LIN {X 0,Y 198.833,Z 382.031,A -85,B 0,C 180,E1 -24400.179,E2 -24400.179} C_VEL
LIN {X 0,Y 188.917,Z 377.763,A -85,B 0,C 180,E1 -24404.769,E2 -24404.769} C_VEL
LIN {X 0,Y 183.38,Z 374.333,A -85,B 0,C 180,E1 -24407.854,E2 -24407.854} C_VEL
LIN {X 0,Y 177.292,Z 368.639,A -85,B 0,C 180,E1 -24412.116,E2 -24412.116} C_VEL
LIN {X 0,Y 173.181,Z 362.778,A -85,B 0,C 180,E1 -24415.87,E2 -24415.87} C_VEL
LIN {X 0,Y 170.579,Z 356.861,A -85,B 0,C 180,E1 -24419.135,E2 -24419.135} C_VEL
LIN {X 0,Y 168.518,Z 348.975,A -85,B 0,C 180,E1 -24422.83,E2 -24422.83} C_VEL
LIN {X 0,Y 167.275,Z 340.992,A -85,B 0,C 180,E1 -24426.029,E2 -24426.029} C_VEL
LIN {X 0,Y 165.67,Z 333.745,A -85,B 0,C 180,E1 -24428.814,E2 -24428.814} C_VEL
LIN {X 0,Y 163.533,Z 326.252,A -85,B 0,C 180,E1 -24431.653,E2 -24431.653} C_VEL
LIN {X 0,Y 160.686,Z 318.576,A -85,B 0,C 180,E1 -24434.641,E2 -24434.641} C_VEL
LIN {X 0,Y 156.368,Z 309.383,A -85,B 0,C 180,E1 -24438.458,E2 -24438.458} C_VEL
LIN {X 0,Y 152.513,Z 302.543,A -85,B 0,C 180,E1 -24441.569,E2 -24441.569} C_VEL
LIN {X 0,Y 150.34,Z 299.173,A -85,B 0,C 180,E1 -24443.332,E2 -24443.332} C_VEL
LIN {X 0,Y 149.453,Z 297.828,A -85,B 0,C 180,E1 -24444.02,E2 -24444.02} C_VEL
LIN {X 0,Y 147.324,Z 294.974,A -85,B 0,C 180,E1 -24445.691,E2 -24445.691} C_VEL
LIN {X 0,Y 146.51,Z 293.362,A -85,B 0,C 180,E1 -24446.457,E2 -24446.457} C_VEL
LIN {X 0,Y 144.109,Z 290.974,A -85,B 0,C 180,E1 -24448.403,E2 -24448.403} C_VEL
LIN {X 0,Y 143.178,Z 288.494,A -85,B 0,C 180,E1 -24449.406,E2 -24449.406} C_VEL
LIN {X 0,Y 143.104,Z 288.159,A -85,B 0,C 180,E1 -24449.593,E2 -24449.593} C_VEL
LIN {X 0,Y 143.128,Z 288.151,A -85,B 0,C 180,E1 -24453.793,E2 -24453.793} C_VEL
LIN {X 0,Y 143.229,Z 288.133,A -85,B 0,C 180,E1 -24459.93,E2 -24459.93} C_VEL
LIN {X 0,Y 143.298,Z 288.126,A -85,B 0,C 180,E1 -24465.823,E2 -24465.823} C_VEL
LIN {X 0,Y 143.521,Z 288.105,A -85,B 0,C 180,E1 -24468.722,E2 -24468.722} C_VEL
LIN {X 0,Y 143.611,Z 288.09,A -85,B 0,C 180,E1 -24471.575,E2 -24471.575} C_VEL
LIN {X 0,Y 144.158,Z 287.993,A -85,B 0,C 180,E1 -24480.016,E2 -24480.016} C_VEL
LIN {X 0,Y 143.622,Z 288.096,A -85,B 0,C 180,E1 -24488.458,E2 -24488.458} C_VEL
LIN {X 0,Y 143.504,Z 288.112,A -85,B 0,C 180,E1 -24491.633,E2 -24491.633} C_VEL
LIN {X 0,Y 143.247,Z 288.145,A -85,B 0,C 180,E1 -24497.136,E2 -24497.136} C_VEL
LIN {X 0,Y 143.35,Z 288.954,A -85,B 0,C 180,E1 -24501.332,E2 -24501.332} C_VEL
LIN {X 0,Y 143.471,Z 290.546,A -85,B 0,C 180,E1 -24508.15,E2 -24508.15} C_VEL
LIN {X 0,Y 143.582,Z 291.452,A -85,B 0,C 180,E1 -24510.74,E2 -24510.74} C_VEL
LIN {X 0,Y 144.635,Z 294.391,A -85,B 0,C 180,E1 -24511.814,E2 -24511.814} C_VEL
LIN {X 0,Y 147.362,Z 297.867,A -85,B 0,C 180,E1 -24514.044,E2 -24514.044} C_VEL
LIN {X 0,Y 148.991,Z 301.335,A -85,B 0,C 180,E1 -24515.523,E2 -24515.523} C_VEL
LIN {X 0,Y 150.405,Z 303.365,A -85,B 0,C 180,E1 -24516.585,E2 -24516.585} C_VEL
LIN {X 0,Y 152.587,Z 307.744,A -85,B 0,C 180,E1 -24518.465,E2 -24518.465} C_VEL
LIN {X 0,Y 155.821,Z 315.822,A -85,B 0,C 180,E1 -24521.485,E2 -24521.485} C_VEL
LIN {X 0,Y 158.01,Z 323.997,A -85,B 0,C 180,E1 -24524.218,E2 -24524.218} C_VEL
LIN {X 0,Y 159.377,Z 333.893,A -85,B 0,C 180,E1 -24527.295,E2 -24527.295} C_VEL
LIN {X 0,Y 159.634,Z 344.227,A -85,B 0,C 180,E1 -24530.573,E2 -24530.573} C_VEL
LIN {X 0,Y 159.227,Z 352.071,A -85,B 0,C 180,E1 -24533.24,E2 -24533.24} C_VEL
LIN {X 0,Y 158.008,Z 360.113,A -85,B 0,C 180,E1 -24536.222,E2 -24536.222} C_VEL
LIN {X 0,Y 154.348,Z 367.945,A -85,B 0,C 180,E1 -24539.187,E2 -24539.187} C_VEL
LIN {X 0,Y 151.04,Z 374.482,A -85,B 0,C 180,E1 -24542.271,E2 -24542.271} C_VEL
LIN {X 0,Y 148.752,Z 378.986,A -85,B 0,C 180,E1 -24544.836,E2 -24544.836} C_VEL
LIN {X 0,Y 145.708,Z 384.478,A -85,B 0,C 180,E1 -24548.793,E2 -24548.793} C_VEL
LIN {X 0,Y 143.303,Z 388.804,A -85,B 0,C 180,E1 -24552.887,E2 -24552.887} C_VEL
LIN {X 0,Y 142.229,Z 391.177,A -85,B 0,C 180,E1 -24555.696,E2 -24555.696} C_VEL
LIN {X 0,Y 141.418,Z 392.982,A -85,B 0,C 180,E1 -24558.534,E2 -24558.534} C_VEL
LIN {X 0,Y 140.571,Z 395.441,A -85,B 0,C 180,E1 -24564.261,E2 -24564.261} C_VEL
LIN {X 0,Y 140.517,Z 396.037,A -85,B 0,C 180,E1 -24567.133,E2 -24567.133} C_VEL
LIN {X 0,Y 140.592,Z 396.196,A -85,B 0,C 180,E1 -24570,E2 -24570} C_VEL
LIN {X 0,Y 140.517,Z 396.037,A -85,B 0,C 180,E1 -24572.867,E2 -24572.867} C_VEL
LIN {X 0,Y 140.57,Z 395.441,A -85,B 0,C 180,E1 -24575.739,E2 -24575.739} C_VEL
LIN {X 0,Y 141.391,Z 392.981,A -85,B 0,C 180,E1 -24581.468,E2 -24581.468} C_VEL
LIN {X 0,Y 142.734,Z 390.024,A -85,B 0,C 180,E1 -24585.712,E2 -24585.712} C_VEL
LIN {X 0,Y 144.826,Z 386.032,A -85,B 0,C 180,E1 -24589.857,E2 -24589.857} C_VEL
LIN {X 0,Y 147.624,Z 380.901,A -85,B 0,C 180,E1 -24593.869,E2 -24593.869} C_VEL
LIN {X 0,Y 150.517,Z 375.641,A -85,B 0,C 180,E1 -24597.08,E2 -24597.08} C_VEL
LIN {X 0,Y 153.589,Z 369.319,A -85,B 0,C 180,E1 -24600.221,E2 -24600.221} C_VEL
LIN {X 0,Y 156.521,Z 363.369,A -85,B 0,C 180,E1 -24602.602,E2 -24602.602} C_VEL
LIN {X 0,Y 157.965,Z 360.112,A -85,B 0,C 180,E1 -24603.788,E2 -24603.788} C_VEL
LIN {X 0,Y 159.233,Z 352.131,A -85,B 0,C 180,E1 -24606.735,E2 -24606.735} C_VEL
LIN {X 0,Y 159.664,Z 342.122,A -85,B 0,C 180,E1 -24610.113,E2 -24610.113} C_VEL
LIN {X 0,Y 159.16,Z 332.099,A -85,B 0,C 180,E1 -24613.25,E2 -24613.25} C_VEL
LIN {X 0,Y 157.994,Z 324.048,A -85,B 0,C 180,E1 -24615.777,E2 -24615.777} C_VEL
LIN {X 0,Y 155.386,Z 314.619,A -85,B 0,C 180,E1 -24618.953,E2 -24618.953} C_VEL
LIN {X 0,Y 152.612,Z 307.745,A -85,B 0,C 180,E1 -24621.523,E2 -24621.523} C_VEL
LIN {X 0,Y 150.325,Z 303.105,A -85,B 0,C 180,E1 -24623.497,E2 -24623.497} C_VEL
LIN {X 0,Y 147.863,Z 299.309,A -85,B 0,C 180,E1 -24625.428,E2 -24625.428} C_VEL
LIN {X 0,Y 147.128,Z 297.299,A -85,B 0,C 180,E1 -24626.188,E2 -24626.188} C_VEL
LIN {X 0,Y 144.635,Z 294.395,A -85,B 0,C 180,E1 -24628.186,E2 -24628.186} C_VEL
LIN {X 0,Y 143.645,Z 291.719,A -85,B 0,C 180,E1 -24629.173,E2 -24629.173} C_VEL
LIN {X 0,Y 143.533,Z 291.167,A -85,B 0,C 180,E1 -24629.452,E2 -24629.452} C_VEL
LIN {X 0,Y 143.494,Z 291.034,A -85,B 0,C 180,E1 -24629.969,E2 -24629.969} C_VEL
LIN {X 0,Y 142.733,Z 290.539,A -85,B 0,C 180,E1 -24632.303,E2 -24632.303} C_VEL
LIN {X 0,Y 141.124,Z 290.215,A -85,B 0,C 180,E1 -24634.61,E2 -24634.61} C_VEL
LIN {X 0,Y 136.565,Z 289.569,A -85,B 0,C 180,E1 -24640.968,E2 -24640.968} C_VEL
LIN {X 0,Y 136.206,Z 289.344,A -85,B 0,C 180,E1 -24642.647,E2 -24642.647} C_VEL
LIN {X 0,Y 136.431,Z 288.991,A -85,B 0,C 180,E1 -24648.161,E2 -24648.161} C_VEL
LIN {X 0,Y 136.549,Z 288.977,A -85,B 0,C 180,E1 -24651.101,E2 -24651.101} C_VEL
LIN {X 0,Y 137.114,Z 288.869,A -85,B 0,C 180,E1 -24659.983,E2 -24659.983} C_VEL
LIN {X 0,Y 136.537,Z 288.968,A -85,B 0,C 180,E1 -24668.865,E2 -24668.865} C_VEL
LIN {X 0,Y 136.402,Z 288.995,A -85,B 0,C 180,E1 -24671.875,E2 -24671.875} C_VEL
LIN {X 0,Y 136.152,Z 289.023,A -85,B 0,C 180,E1 -24678.023,E2 -24678.023} C_VEL
LIN {X 0,Y 136.133,Z 289.025,A -85,B 0,C 180,E1 -24681.682,E2 -24681.682} C_VEL
LIN {X 0,Y 136.043,Z 289.072,A -85,B 0,C 180,E1 -24685.103,E2 -24685.103} C_VEL
LIN {X 0,Y 136.787,Z 291.353,A -85,B 0,C 180,E1 -24686.181,E2 -24686.181} C_VEL
LIN {X 0,Y 138.729,Z 293.698,A -85,B 0,C 180,E1 -24688.314,E2 -24688.314} C_VEL
LIN {X 0,Y 140.046,Z 294.733,A -85,B 0,C 180,E1 -24689.534,E2 -24689.534} C_VEL
LIN {X 0,Y 141.538,Z 297.697,A -85,B 0,C 180,E1 -24691.195,E2 -24691.195} C_VEL
LIN {X 0,Y 143.238,Z 299.416,A -85,B 0,C 180,E1 -24692.643,E2 -24692.643} C_VEL
LIN {X 0,Y 145.196,Z 302.88,A -85,B 0,C 180,E1 -24694.63,E2 -24694.63} C_VEL
LIN {X 0,Y 146.612,Z 305.028,A -85,B 0,C 180,E1 -24695.937,E2 -24695.937} C_VEL
LIN {X 0,Y 150.135,Z 311.111,A -85,B 0,C 180,E1 -24699.156,E2 -24699.156} C_VEL
LIN {X 0,Y 153.511,Z 318.085,A -85,B 0,C 180,E1 -24702.452,E2 -24702.452} C_VEL
LIN {X 0,Y 156.589,Z 325.893,A -85,B 0,C 180,E1 -24705.873,E2 -24705.873} C_VEL
LIN {X 0,Y 159.072,Z 334.163,A -85,B 0,C 180,E1 -24709.305,E2 -24709.305} C_VEL
LIN {X 0,Y 161.027,Z 343.496,A -85,B 0,C 180,E1 -24713.145,E2 -24713.145} C_VEL
LIN {X 0,Y 162.338,Z 353.017,A -85,B 0,C 180,E1 -24717.353,E2 -24717.353} C_VEL
LIN {X 0,Y 164.456,Z 360.598,A -85,B 0,C 180,E1 -24721.389,E2 -24721.389} C_VEL
LIN {X 0,Y 167.431,Z 366.658,A -85,B 0,C 180,E1 -24725.182,E2 -24725.182} C_VEL
LIN {X 0,Y 172.361,Z 372.655,A -85,B 0,C 180,E1 -24729.64,E2 -24729.64} C_VEL
LIN {X 0,Y 178.939,Z 377.595,A -85,B 0,C 180,E1 -24734.042,E2 -24734.042} C_VEL
LIN {X 0,Y 186.682,Z 381.335,A -85,B 0,C 180,E1 -24738.108,E2 -24738.108} C_VEL
LIN {X 0,Y 198.202,Z 384.674,A -85,B 0,C 180,E1 -24743.013,E2 -24743.013} C_VEL
LIN {X 0,Y 206.464,Z 385.982,A -85,B 0,C 180,E1 -24746.096,E2 -24746.096} C_VEL
LIN {X 0,Y 211.895,Z 386.401,A -85,B 0,C 180,E1 -24748.099,E2 -24748.099} C_VEL
LIN {X 0,Y 216.225,Z 386.453,A -85,B 0,C 180,E1 -24750,E2 -24750} C_VEL
LIN {X 0,Y 210.951,Z 386.331,A -85,B 0,C 180,E1 -24752.266,E2 -24752.266} C_VEL
LIN {X 0,Y 204.438,Z 385.724,A -85,B 0,C 180,E1 -24754.674,E2 -24754.674} C_VEL
LIN {X 0,Y 194.909,Z 383.923,A -85,B 0,C 180,E1 -24758.293,E2 -24758.293} C_VEL
LIN {X 0,Y 186.681,Z 381.337,A -85,B 0,C 180,E1 -24761.89,E2 -24761.89} C_VEL
LIN {X 0,Y 178.922,Z 377.596,A -85,B 0,C 180,E1 -24765.959,E2 -24765.959} C_VEL
LIN {X 0,Y 174.508,Z 374.586,A -85,B 0,C 180,E1 -24768.795,E2 -24768.795} C_VEL
LIN {X 0,Y 169.168,Z 369.205,A -85,B 0,C 180,E1 -24773.05,E2 -24773.05} C_VEL
LIN {X 0,Y 165.569,Z 363.332,A -85,B 0,C 180,E1 -24776.988,E2 -24776.988} C_VEL
LIN {X 0,Y 163.267,Z 357,A -85,B 0,C 180,E1 -24780.614,E2 -24780.614} C_VEL
LIN {X 0,Y 161.755,Z 349.195,A -85,B 0,C 180,E1 -24784.39,E2 -24784.39} C_VEL
LIN {X 0,Y 160.621,Z 341.221,A -85,B 0,C 180,E1 -24787.775,E2 -24787.775} C_VEL
LIN {X 0,Y 159.063,Z 334.194,A -85,B 0,C 180,E1 -24790.689,E2 -24790.689} C_VEL
LIN {X 0,Y 156.583,Z 325.908,A -85,B 0,C 180,E1 -24794.125,E2 -24794.125} C_VEL
LIN {X 0,Y 153.513,Z 318.079,A -85,B 0,C 180,E1 -24797.549,E2 -24797.549} C_VEL
LIN {X 0,Y 148.768,Z 308.578,A -85,B 0,C 180,E1 -24802.134,E2 -24802.134} C_VEL
LIN {X 0,Y 145.951,Z 303.772,A -85,B 0,C 180,E1 -24804.724,E2 -24804.724} C_VEL
LIN {X 0,Y 143.783,Z 300.431,A -85,B 0,C 180,E1 -24806.809,E2 -24806.809} C_VEL
LIN {X 0,Y 143.042,Z 299.241,A -85,B 0,C 180,E1 -24807.516,E2 -24807.516} C_VEL
LIN {X 0,Y 140.791,Z 296.525,A -85,B 0,C 180,E1 -24809.559,E2 -24809.559} C_VEL
LIN {X 0,Y 139.902,Z 294.502,A -85,B 0,C 180,E1 -24810.621,E2 -24810.621} C_VEL
LIN {X 0,Y 137.212,Z 292.058,A -85,B 0,C 180,E1 -24813.292,E2 -24813.292} C_VEL
LIN {X 0,Y 136.155,Z 289.643,A -85,B 0,C 180,E1 -24814.714,E2 -24814.714} C_VEL
LIN {X 0,Y 136.04,Z 289.029,A -85,B 0,C 180,E1 -24814.998,E2 -24814.998} C_VEL
LIN {X 0,Y 136.17,Z 289.017,A -85,B 0,C 180,E1 -24818.841,E2 -24818.841} C_VEL
LIN {X 0,Y 136.214,Z 289.007,A -85,B 0,C 180,E1 -24825.069,E2 -24825.069} C_VEL
LIN {X 0,Y 136.414,Z 288.993,A -85,B 0,C 180,E1 -24828.195,E2 -24828.195} C_VEL
LIN {X 0,Y 136.537,Z 288.968,A -85,B 0,C 180,E1 -24831.135,E2 -24831.135} C_VEL
LIN {X 0,Y 137.114,Z 288.869,A -85,B 0,C 180,E1 -24840.017,E2 -24840.017} C_VEL
LIN {X 0,Y 136.549,Z 288.976,A -85,B 0,C 180,E1 -24848.899,E2 -24848.899} C_VEL
LIN {X 0,Y 136.419,Z 288.996,A -85,B 0,C 180,E1 -24851.909,E2 -24851.909} C_VEL
LIN {X 0,Y 136.231,Z 289.018,A -85,B 0,C 180,E1 -24854.965,E2 -24854.965} C_VEL
LIN {X 0,Y 136.333,Z 290.022,A -85,B 0,C 180,E1 -24861.17,E2 -24861.17} C_VEL
LIN {X 0,Y 136.354,Z 291.117,A -85,B 0,C 180,E1 -24865.182,E2 -24865.182} C_VEL
LIN {X 0,Y 137.516,Z 294.167,A -85,B 0,C 180,E1 -24866.683,E2 -24866.683} C_VEL
LIN {X 0,Y 140.455,Z 297.698,A -85,B 0,C 180,E1 -24869.655,E2 -24869.655} C_VEL
LIN {X 0,Y 141.779,Z 300.798,A -85,B 0,C 180,E1 -24871.174,E2 -24871.174} C_VEL
LIN {X 0,Y 143.825,Z 303.593,A -85,B 0,C 180,E1 -24872.989,E2 -24872.989} C_VEL
LIN {X 0,Y 145.659,Z 307.426,A -85,B 0,C 180,E1 -24874.893,E2 -24874.893} C_VEL
LIN {X 0,Y 148.709,Z 313.993,A -85,B 0,C 180,E1 -24877.924,E2 -24877.924} C_VEL
LIN {X 0,Y 150.498,Z 318.822,A -85,B 0,C 180,E1 -24879.967,E2 -24879.967} C_VEL
LIN {X 0,Y 152.465,Z 326.73,A -85,B 0,C 180,E1 -24882.855,E2 -24882.855} C_VEL
LIN {X 0,Y 153.531,Z 336.179,A -85,B 0,C 180,E1 -24886.06,E2 -24886.06} C_VEL
LIN {X 0,Y 153.542,Z 344.648,A -85,B 0,C 180,E1 -24888.92,E2 -24888.92} C_VEL
LIN {X 0,Y 152.971,Z 353.077,A -85,B 0,C 180,E1 -24891.993,E2 -24891.993} C_VEL
LIN {X 0,Y 151.935,Z 359.911,A -85,B 0,C 180,E1 -24894.676,E2 -24894.676} C_VEL
LIN {X 0,Y 150.593,Z 363.175,A -85,B 0,C 180,E1 -24895.943,E2 -24895.943} C_VEL
LIN {X 0,Y 147.532,Z 369.125,A -85,B 0,C 180,E1 -24898.399,E2 -24898.399} C_VEL
LIN {X 0,Y 144.18,Z 375.373,A -85,B 0,C 180,E1 -24901.577,E2 -24901.577} C_VEL
LIN {X 0,Y 142.356,Z 378.792,A -85,B 0,C 180,E1 -24903.621,E2 -24903.621} C_VEL
LIN {X 0,Y 139.086,Z 384.282,A -85,B 0,C 180,E1 -24907.73,E2 -24907.73} C_VEL
LIN {X 0,Y 136.496,Z 388.608,A -85,B 0,C 180,E1 -24912.006,E2 -24912.006} C_VEL
LIN {X 0,Y 135.337,Z 390.981,A -85,B 0,C 180,E1 -24914.951,E2 -24914.951} C_VEL
LIN {X 0,Y 134.454,Z 392.787,A -85,B 0,C 180,E1 -24917.932,E2 -24917.932} C_VEL
LIN {X 0,Y 133.49,Z 395.245,A -85,B 0,C 180,E1 -24923.956,E2 -24923.956} C_VEL
LIN {X 0,Y 133.428,Z 395.842,A -85,B 0,C 180,E1 -24926.981,E2 -24926.981} C_VEL
LIN {X 0,Y 133.506,Z 396.002,A -85,B 0,C 180,E1 -24930,E2 -24930} C_VEL
LIN {X 0,Y 133.428,Z 395.842,A -85,B 0,C 180,E1 -24933.019,E2 -24933.019} C_VEL
LIN {X 0,Y 133.487,Z 395.245,A -85,B 0,C 180,E1 -24936.044,E2 -24936.044} C_VEL
LIN {X 0,Y 134.402,Z 392.785,A -85,B 0,C 180,E1 -24942.073,E2 -24942.073} C_VEL
LIN {X 0,Y 135.876,Z 389.828,A -85,B 0,C 180,E1 -24946.527,E2 -24946.527} C_VEL
LIN {X 0,Y 138.14,Z 385.836,A -85,B 0,C 180,E1 -24950.862,E2 -24950.862} C_VEL
LIN {X 0,Y 141.14,Z 380.705,A -85,B 0,C 180,E1 -24955.039,E2 -24955.039} C_VEL
LIN {X 0,Y 143.578,Z 376.601,A -85,B 0,C 180,E1 -24957.71,E2 -24957.71} C_VEL
LIN {X 0,Y 146.701,Z 370.637,A -85,B 0,C 180,E1 -24960.916,E2 -24960.916} C_VEL
LIN {X 0,Y 149.774,Z 364.801,A -85,B 0,C 180,E1 -24963.459,E2 -24963.459} C_VEL
LIN {X 0,Y 151.347,Z 361.546,A -85,B 0,C 180,E1 -24964.669,E2 -24964.669} C_VEL
LIN {X 0,Y 152.559,Z 356.204,A -85,B 0,C 180,E1 -24966.788,E2 -24966.788} C_VEL
LIN {X 0,Y 153.312,Z 349.59,A -85,B 0,C 180,E1 -24969.307,E2 -24969.307} C_VEL
LIN {X 0,Y 153.641,Z 341.086,A -85,B 0,C 180,E1 -24972.296,E2 -24972.296} C_VEL
LIN {X 0,Y 153.177,Z 332.345,A -85,B 0,C 180,E1 -24975.259,E2 -24975.259} C_VEL
LIN {X 0,Y 152.046,Z 324.717,A -85,B 0,C 180,E1 -24977.896,E2 -24977.896} C_VEL
LIN {X 0,Y 149.955,Z 317.139,A -85,B 0,C 180,E1 -24980.711,E2 -24980.711} C_VEL
LIN {X 0,Y 147.367,Z 311.006,A -85,B 0,C 180,E1 -24983.39,E2 -24983.39} C_VEL
LIN {X 0,Y 145.659,Z 307.426,A -85,B 0,C 180,E1 -24985.107,E2 -24985.107} C_VEL
LIN {X 0,Y 143.7,Z 303.242,A -85,B 0,C 180,E1 -24987.15,E2 -24987.15} C_VEL
LIN {X 0,Y 141.122,Z 299.619,A -85,B 0,C 180,E1 -24989.496,E2 -24989.496} C_VEL
LIN {X 0,Y 140.307,Z 297.25,A -85,B 0,C 180,E1 -24990.542,E2 -24990.542} C_VEL
LIN {X 0,Y 137.67,Z 294.405,A -85,B 0,C 180,E1 -24993.145,E2 -24993.145} C_VEL
LIN {X 0,Y 136.455,Z 291.617,A -85,B 0,C 180,E1 -24994.634,E2 -24994.634} C_VEL
LIN {X 0,Y 136.302,Z 290.837,A -85,B 0,C 180,E1 -24995.011,E2 -24995.011} C_VEL
LIN {X 0,Y 136.332,Z 290.021,A -85,B 0,C 180,E1 -24998.83,E2 -24998.83} C_VEL
LIN {X 0,Y 136.206,Z 289.344,A -85,B 0,C 180,E1 -25002.647,E2 -25002.647} C_VEL
LIN {X 0,Y 135.847,Z 289.206,A -85,B 0,C 180,E1 -25004.298,E2 -25004.298} C_VEL
LIN {X 0,Y 134.501,Z 289.254,A -85,B 0,C 180,E1 -25006.747,E2 -25006.747} C_VEL
LIN {X 0,Y 129.726,Z 289.826,A -85,B 0,C 180,E1 -25014.303,E2 -25014.303} C_VEL
LIN {X 0,Y 129.554,Z 289.843,A -85,B 0,C 180,E1 -25016.075,E2 -25016.075} C_VEL
LIN {X 0,Y 130.069,Z 289.745,A -85,B 0,C 180,E1 -25019.982,E2 -25019.982} C_VEL
LIN {X 0,Y 129.46,Z 289.848,A -85,B 0,C 180,E1 -25029.354,E2 -25029.354} C_VEL
LIN {X 0,Y 129.286,Z 289.88,A -85,B 0,C 180,E1 -25032.539,E2 -25032.539} C_VEL
LIN {X 0,Y 129.107,Z 289.98,A -85,B 0,C 180,E1 -25037.503,E2 -25037.503} C_VEL
LIN {X 0,Y 129.822,Z 292.286,A -85,B 0,C 180,E1 -25039.139,E2 -25039.139} C_VEL
LIN {X 0,Y 132.315,Z 295.053,A -85,B 0,C 180,E1 -25042.897,E2 -25042.897} C_VEL
LIN {X 0,Y 133.37,Z 295.869,A -85,B 0,C 180,E1 -25044.186,E2 -25044.186} C_VEL
LIN {X 0,Y 134.903,Z 298.878,A -85,B 0,C 180,E1 -25046.367,E2 -25046.367} C_VEL
LIN {X 0,Y 136.105,Z 300.097,A -85,B 0,C 180,E1 -25047.671,E2 -25047.671} C_VEL
LIN {X 0,Y 138.406,Z 303.836,A -85,B 0,C 180,E1 -25050.494,E2 -25050.494} C_VEL
LIN {X 0,Y 139.75,Z 305.365,A -85,B 0,C 180,E1 -25051.851,E2 -25051.851} C_VEL
LIN {X 0,Y 142.892,Z 310.892,A -85,B 0,C 180,E1 -25055.271,E2 -25055.271} C_VEL
LIN {X 0,Y 146.767,Z 318.467,A -85,B 0,C 180,E1 -25059.516,E2 -25059.516} C_VEL
LIN {X 0,Y 150.012,Z 326.528,A -85,B 0,C 180,E1 -25063.499,E2 -25063.499} C_VEL
LIN {X 0,Y 152.635,Z 335.088,A -85,B 0,C 180,E1 -25067.425,E2 -25067.425} C_VEL
LIN {X 0,Y 154.476,Z 344.226,A -85,B 0,C 180,E1 -25071.493,E2 -25071.493} C_VEL
LIN {X 0,Y 155.558,Z 353.811,A -85,B 0,C 180,E1 -25076.02,E2 -25076.02} C_VEL
LIN {X 0,Y 157.061,Z 360.881,A -85,B 0,C 180,E1 -25079.936,E2 -25079.936} C_VEL
LIN {X 0,Y 159.512,Z 366.893,A -85,B 0,C 180,E1 -25083.859,E2 -25083.859} C_VEL
LIN {X 0,Y 162.33,Z 371.201,A -85,B 0,C 180,E1 -25087.068,E2 -25087.068} C_VEL
LIN {X 0,Y 167.72,Z 376.343,A -85,B 0,C 180,E1 -25091.638,E2 -25091.638} C_VEL
LIN {X 0,Y 174.6,Z 380.419,A -85,B 0,C 180,E1 -25096.025,E2 -25096.025} C_VEL
LIN {X 0,Y 179.759,Z 382.564,A -85,B 0,C 180,E1 -25098.727,E2 -25098.727} C_VEL
LIN {X 0,Y 185.256,Z 384.185,A -85,B 0,C 180,E1 -25101.272,E2 -25101.272} C_VEL
LIN {X 0,Y 197.215,Z 386.257,A -85,B 0,C 180,E1 -25105.984,E2 -25105.984} C_VEL
LIN {X 0,Y 203.837,Z 386.713,A -85,B 0,C 180,E1 -25108.411,E2 -25108.411} C_VEL
LIN {X 0,Y 207.848,Z 386.678,A -85,B 0,C 180,E1 -25110,E2 -25110} C_VEL
LIN {X 0,Y 202.845,Z 386.648,A -85,B 0,C 180,E1 -25111.985,E2 -25111.985} C_VEL
LIN {X 0,Y 197.063,Z 386.239,A -85,B 0,C 180,E1 -25114.09,E2 -25114.09} C_VEL
LIN {X 0,Y 184.893,Z 384.086,A -85,B 0,C 180,E1 -25118.882,E2 -25118.882} C_VEL
LIN {X 0,Y 179.255,Z 382.403,A -85,B 0,C 180,E1 -25121.513,E2 -25121.513} C_VEL
LIN {X 0,Y 172.118,Z 379.251,A -85,B 0,C 180,E1 -25125.404,E2 -25125.404} C_VEL
LIN {X 0,Y 165.001,Z 374.048,A -85,B 0,C 180,E1 -25130.486,E2 -25130.486} C_VEL
LIN {X 0,Y 160.608,Z 368.801,A -85,B 0,C 180,E1 -25134.756,E2 -25134.756} C_VEL
LIN {X 0,Y 157.716,Z 362.924,A -85,B 0,C 180,E1 -25138.8,E2 -25138.8} C_VEL
LIN {X 0,Y 155.92,Z 356.159,A -85,B 0,C 180,E1 -25142.743,E2 -25142.743} C_VEL
LIN {X 0,Y 155.105,Z 349.419,A -85,B 0,C 180,E1 -25146.088,E2 -25146.088} C_VEL
LIN {X 0,Y 154.16,Z 342.598,A -85,B 0,C 180,E1 -25149.222,E2 -25149.222} C_VEL
LIN {X 0,Y 152.613,Z 335.138,A -85,B 0,C 180,E1 -25152.565,E2 -25152.565} C_VEL
LIN {X 0,Y 149.993,Z 326.569,A -85,B 0,C 180,E1 -25156.497,E2 -25156.497} C_VEL
LIN {X 0,Y 146.747,Z 318.486,A -85,B 0,C 180,E1 -25160.488,E2 -25160.488} C_VEL
LIN {X 0,Y 142.142,Z 309.384,A -85,B 0,C 180,E1 -25165.591,E2 -25165.591} C_VEL
LIN {X 0,Y 139.747,Z 305.376,A -85,B 0,C 180,E1 -25168.148,E2 -25168.148} C_VEL
LIN {X 0,Y 138.011,Z 303.248,A -85,B 0,C 180,E1 -25169.96,E2 -25169.96} C_VEL
LIN {X 0,Y 137.305,Z 301.765,A -85,B 0,C 180,E1 -25170.925,E2 -25170.925} C_VEL
LIN {X 0,Y 133.875,Z 297.204,A -85,B 0,C 180,E1 -25174.981,E2 -25174.981} C_VEL
LIN {X 0,Y 133.183,Z 295.532,A -85,B 0,C 180,E1 -25176.088,E2 -25176.088} C_VEL
LIN {X 0,Y 130.456,Z 293.291,A -85,B 0,C 180,E1 -25179.729,E2 -25179.729} C_VEL
LIN {X 0,Y 129.378,Z 291.131,A -85,B 0,C 180,E1 -25181.819,E2 -25181.819} C_VEL
LIN {X 0,Y 129.093,Z 289.905,A -85,B 0,C 180,E1 -25182.597,E2 -25182.597} C_VEL
LIN {X 0,Y 129.332,Z 289.875,A -85,B 0,C 180,E1 -25187.99,E2 -25187.99} C_VEL
LIN {X 0,Y 129.46,Z 289.848,A -85,B 0,C 180,E1 -25190.646,E2 -25190.646} C_VEL
LIN {X 0,Y 130.069,Z 289.745,A -85,B 0,C 180,E1 -25200.018,E2 -25200.018} C_VEL
LIN {X 0,Y 129.472,Z 289.859,A -85,B 0,C 180,E1 -25209.39,E2 -25209.39} C_VEL
LIN {X 0,Y 129.303,Z 289.881,A -85,B 0,C 180,E1 -25212.575,E2 -25212.575} C_VEL
LIN {X 0,Y 129.205,Z 290.497,A -85,B 0,C 180,E1 -25217.222,E2 -25217.222} C_VEL
LIN {X 0,Y 130.238,Z 293.491,A -85,B 0,C 180,E1 -25219.318,E2 -25219.318} C_VEL
LIN {X 0,Y 133.21,Z 296.96,A -85,B 0,C 180,E1 -25223.533,E2 -25223.533} C_VEL
LIN {X 0,Y 133.732,Z 297.833,A -85,B 0,C 180,E1 -25224.258,E2 -25224.258} C_VEL
LIN {X 0,Y 135.11,Z 300.973,A -85,B 0,C 180,E1 -25226.258,E2 -25226.258} C_VEL
LIN {X 0,Y 137.254,Z 303.752,A -85,B 0,C 180,E1 -25228.601,E2 -25228.601} C_VEL
LIN {X 0,Y 138.7,Z 307.073,A -85,B 0,C 180,E1 -25230.528,E2 -25230.528} C_VEL
LIN {X 0,Y 139.948,Z 308.871,A -85,B 0,C 180,E1 -25231.839,E2 -25231.839} C_VEL
LIN {X 0,Y 143.477,Z 316.875,A -85,B 0,C 180,E1 -25236.019,E2 -25236.019} C_VEL
LIN {X 0,Y 145.919,Z 324.159,A -85,B 0,C 180,E1 -25239.281,E2 -25239.281} C_VEL
LIN {X 0,Y 147.296,Z 331.991,A -85,B 0,C 180,E1 -25242.346,E2 -25242.346} C_VEL
LIN {X 0,Y 147.759,Z 340.702,A -85,B 0,C 180,E1 -25245.536,E2 -25245.536} C_VEL
LIN {X 0,Y 147.189,Z 351.113,A -85,B 0,C 180,E1 -25249.416,E2 -25249.416} C_VEL
LIN {X 0,Y 145.819,Z 359.704,A -85,B 0,C 180,E1 -25252.955,E2 -25252.955} C_VEL
LIN {X 0,Y 145.444,Z 361.347,A -85,B 0,C 180,E1 -25253.707,E2 -25253.707} C_VEL
LIN {X 0,Y 142.281,Z 367.553,A -85,B 0,C 180,E1 -25256.242,E2 -25256.242} C_VEL
LIN {X 0,Y 138.243,Z 374.611,A -85,B 0,C 180,E1 -25259.825,E2 -25259.825} C_VEL
LIN {X 0,Y 136.007,Z 378.596,A -85,B 0,C 180,E1 -25262.286,E2 -25262.286} C_VEL
LIN {X 0,Y 132.516,Z 384.087,A -85,B 0,C 180,E1 -25266.562,E2 -25266.562} C_VEL
LIN {X 0,Y 129.729,Z 388.412,A -85,B 0,C 180,E1 -25271.032,E2 -25271.032} C_VEL
LIN {X 0,Y 128.456,Z 390.786,A -85,B 0,C 180,E1 -25274.124,E2 -25274.124} C_VEL
LIN {X 0,Y 127.483,Z 392.591,A -85,B 0,C 180,E1 -25277.261,E2 -25277.261} C_VEL
LIN {X 0,Y 126.433,Z 395.051,A -85,B 0,C 180,E1 -25283.617,E2 -25283.617} C_VEL
LIN {X 0,Y 126.334,Z 395.647,A -85,B 0,C 180,E1 -25286.811,E2 -25286.811} C_VEL
LIN {X 0,Y 126.422,Z 395.807,A -85,B 0,C 180,E1 -25290,E2 -25290} C_VEL
LIN {X 0,Y 126.334,Z 395.647,A -85,B 0,C 180,E1 -25293.189,E2 -25293.189} C_VEL
LIN {X 0,Y 126.428,Z 395.051,A -85,B 0,C 180,E1 -25296.383,E2 -25296.383} C_VEL
LIN {X 0,Y 127.442,Z 392.59,A -85,B 0,C 180,E1 -25302.743,E2 -25302.743} C_VEL
LIN {X 0,Y 129.033,Z 389.632,A -85,B 0,C 180,E1 -25307.431,E2 -25307.431} C_VEL
LIN {X 0,Y 131.505,Z 385.641,A -85,B 0,C 180,E1 -25311.968,E2 -25311.968} C_VEL
LIN {X 0,Y 134.728,Z 380.51,A -85,B 0,C 180,E1 -25316.32,E2 -25316.32} C_VEL
LIN {X 0,Y 137.794,Z 375.506,A -85,B 0,C 180,E1 -25319.632,E2 -25319.632} C_VEL
LIN {X 0,Y 141.452,Z 368.928,A -85,B 0,C 180,E1 -25323.128,E2 -25323.128} C_VEL
LIN {X 0,Y 144.718,Z 362.978,A -85,B 0,C 180,E1 -25325.644,E2 -25325.644} C_VEL
LIN {X 0,Y 145.828,Z 359.704,A -85,B 0,C 180,E1 -25327.042,E2 -25327.042} C_VEL
LIN {X 0,Y 147.194,Z 351.119,A -85,B 0,C 180,E1 -25330.579,E2 -25330.579} C_VEL
LIN {X 0,Y 147.743,Z 342.457,A -85,B 0,C 180,E1 -25333.854,E2 -25333.854} C_VEL
LIN {X 0,Y 147.419,Z 332.99,A -85,B 0,C 180,E1 -25337.298,E2 -25337.298} C_VEL
LIN {X 0,Y 146.127,Z 325.19,A -85,B 0,C 180,E1 -25340.309,E2 -25340.309} C_VEL
LIN {X 0,Y 144.548,Z 319.915,A -85,B 0,C 180,E1 -25342.555,E2 -25342.555} C_VEL
LIN {X 0,Y 141.784,Z 312.908,A -85,B 0,C 180,E1 -25346.013,E2 -25346.013} C_VEL
LIN {X 0,Y 139.951,Z 308.861,A -85,B 0,C 180,E1 -25348.162,E2 -25348.162} C_VEL
LIN {X 0,Y 138.069,Z 305.935,A -85,B 0,C 180,E1 -25350.227,E2 -25350.227} C_VEL
LIN {X 0,Y 136.883,Z 303.054,A -85,B 0,C 180,E1 -25351.837,E2 -25351.837} C_VEL
LIN {X 0,Y 134.418,Z 299.743,A -85,B 0,C 180,E1 -25354.637,E2 -25354.637} C_VEL
LIN {X 0,Y 133.367,Z 297.052,A -85,B 0,C 180,E1 -25356.291,E2 -25356.291} C_VEL
LIN {X 0,Y 130.462,Z 293.864,A -85,B 0,C 180,E1 -25360.307,E2 -25360.307} C_VEL
LIN {X 0,Y 129.31,Z 290.975,A -85,B 0,C 180,E1 -25362.487,E2 -25362.487} C_VEL
LIN {X 0,Y 129.197,Z 290.396,A -85,B 0,C 180,E1 -25362.981,E2 -25362.981} C_VEL
LIN {X 0,Y 129.349,Z 289.873,A -85,B 0,C 180,E1 -25367.955,E2 -25367.955} C_VEL
LIN {X 0,Y 129.472,Z 289.858,A -85,B 0,C 180,E1 -25370.61,E2 -25370.61} C_VEL
LIN {X 0,Y 129.554,Z 289.843,A -85,B 0,C 180,E1 -25376.075,E2 -25376.075} C_VEL
LIN {X 0,Y 129.369,Z 289.959,A -85,B 0,C 180,E1 -25377.809,E2 -25377.809} C_VEL
LIN {X 0,Y 128.678,Z 290.292,A -85,B 0,C 180,E1 -25379.523,E2 -25379.523} C_VEL
LIN {X 0,Y 126.534,Z 291.426,A -85,B 0,C 180,E1 -25382.925,E2 -25382.925} C_VEL
LIN {X 0,Y 124.512,Z 292.956,A -85,B 0,C 180,E1 -25386.434,E2 -25386.434} C_VEL
LIN {X 0,Y 123.98,Z 294.183,A -85,B 0,C 180,E1 -25389.143,E2 -25389.143} C_VEL
LIN {X 0,Y 124.117,Z 294.583,A -85,B 0,C 180,E1 -25390.05,E2 -25390.05} C_VEL
LIN {X 0,Y 126.873,Z 296.873,A -85,B 0,C 180,E1 -25396.679,E2 -25396.679} C_VEL
LIN {X 0,Y 127.959,Z 299.534,A -85,B 0,C 180,E1 -25399.22,E2 -25399.22} C_VEL
LIN {X 0,Y 130.612,Z 302.221,A -85,B 0,C 180,E1 -25403.269,E2 -25403.269} C_VEL
LIN {X 0,Y 131.69,Z 304.678,A -85,B 0,C 180,E1 -25405.252,E2 -25405.252} C_VEL
LIN {X 0,Y 133.881,Z 307.66,A -85,B 0,C 180,E1 -25408.172,E2 -25408.172} C_VEL
LIN {X 0,Y 135.016,Z 309.776,A -85,B 0,C 180,E1 -25409.714,E2 -25409.714} C_VEL
LIN {X 0,Y 136.177,Z 311.215,A -85,B 0,C 180,E1 -25411.048,E2 -25411.048} C_VEL
LIN {X 0,Y 140.067,Z 318.886,A -85,B 0,C 180,E1 -25416.103,E2 -25416.103} C_VEL
LIN {X 0,Y 143.332,Z 326.739,A -85,B 0,C 180,E1 -25420.585,E2 -25420.585} C_VEL
LIN {X 0,Y 145.682,Z 334.008,A -85,B 0,C 180,E1 -25424.36,E2 -25424.36} C_VEL
LIN {X 0,Y 147.138,Z 339.944,A -85,B 0,C 180,E1 -25427.301,E2 -25427.301} C_VEL
LIN {X 0,Y 148.249,Z 346.942,A -85,B 0,C 180,E1 -25430.697,E2 -25430.697} C_VEL
LIN {X 0,Y 148.881,Z 354.015,A -85,B 0,C 180,E1 -25434.259,E2 -25434.259} C_VEL
LIN {X 0,Y 149.86,Z 361.208,A -85,B 0,C 180,E1 -25438.387,E2 -25438.387} C_VEL
LIN {X 0,Y 151.806,Z 367.128,A -85,B 0,C 180,E1 -25442.423,E2 -25442.423} C_VEL
LIN {X 0,Y 154.171,Z 371.441,A -85,B 0,C 180,E1 -25445.779,E2 -25445.779} C_VEL
LIN {X 0,Y 159.196,Z 376.79,A -85,B 0,C 180,E1 -25450.798,E2 -25450.798} C_VEL
LIN {X 0,Y 165.343,Z 380.676,A -85,B 0,C 180,E1 -25455.225,E2 -25455.225} C_VEL
LIN {X 0,Y 171.834,Z 383.315,A -85,B 0,C 180,E1 -25458.902,E2 -25458.902} C_VEL
LIN {X 0,Y 177.531,Z 384.931,A -85,B 0,C 180,E1 -25461.648,E2 -25461.648} C_VEL
LIN {X 0,Y 187.378,Z 386.503,A -85,B 0,C 180,E1 -25465.698,E2 -25465.698} C_VEL
LIN {X 0,Y 196.753,Z 386.976,A -85,B 0,C 180,E1 -25469.128,E2 -25469.128} C_VEL
LIN {X 0,Y 199.09,Z 386.914,A -85,B 0,C 180,E1 -25470,E2 -25470} C_VEL
LIN {X 0,Y 193.477,Z 386.904,A -85,B 0,C 180,E1 -25472.082,E2 -25472.082} C_VEL
LIN {X 0,Y 183.608,Z 386.001,A -85,B 0,C 180,E1 -25475.778,E2 -25475.778} C_VEL
LIN {X 0,Y 175.692,Z 384.445,A -85,B 0,C 180,E1 -25479.207,E2 -25479.207} C_VEL
LIN {X 0,Y 170.316,Z 382.829,A -85,B 0,C 180,E1 -25481.907,E2 -25481.907} C_VEL
LIN {X 0,Y 161.791,Z 378.675,A -85,B 0,C 180,E1 -25487.188,E2 -25487.188} C_VEL
LIN {X 0,Y 157.276,Z 375.081,A -85,B 0,C 180,E1 -25490.945,E2 -25490.945} C_VEL
LIN {X 0,Y 152.875,Z 369.348,A -85,B 0,C 180,E1 -25495.894,E2 -25495.894} C_VEL
LIN {X 0,Y 150.439,Z 363.485,A -85,B 0,C 180,E1 -25500.144,E2 -25500.144} C_VEL
LIN {X 0,Y 149.23,Z 357.687,A -85,B 0,C 180,E1 -25503.74,E2 -25503.74} C_VEL
LIN {X 0,Y 148.67,Z 351.013,A -85,B 0,C 180,E1 -25507.292,E2 -25507.292} C_VEL
LIN {X 0,Y 147.9,Z 344.521,A -85,B 0,C 180,E1 -25510.538,E2 -25510.538} C_VEL
LIN {X 0,Y 146.512,Z 337.423,A -85,B 0,C 180,E1 -25514.011,E2 -25514.011} C_VEL
LIN {X 0,Y 144.355,Z 329.753,A -85,B 0,C 180,E1 -25517.847,E2 -25517.847} C_VEL
LIN {X 0,Y 141.557,Z 322.336,A -85,B 0,C 180,E1 -25521.845,E2 -25521.845} C_VEL
LIN {X 0,Y 138.326,Z 315.442,A -85,B 0,C 180,E1 -25526.044,E2 -25526.044} C_VEL
LIN {X 0,Y 136.178,Z 311.213,A -85,B 0,C 180,E1 -25528.952,E2 -25528.952} C_VEL
LIN {X 0,Y 134.424,Z 308.783,A -85,B 0,C 180,E1 -25531.044,E2 -25531.044} C_VEL
LIN {X 0,Y 133.896,Z 307.611,A -85,B 0,C 180,E1 -25531.832,E2 -25531.832} C_VEL
LIN {X 0,Y 131.129,Z 303.66,A -85,B 0,C 180,E1 -25535.66,E2 -25535.66} C_VEL
LIN {X 0,Y 130.613,Z 302.218,A -85,B 0,C 180,E1 -25536.731,E2 -25536.731} C_VEL
LIN {X 0,Y 127.66,Z 299.032,A -85,B 0,C 180,E1 -25541.358,E2 -25541.358} C_VEL
LIN {X 0,Y 126.813,Z 296.617,A -85,B 0,C 180,E1 -25543.52,E2 -25543.52} C_VEL
LIN {X 0,Y 124.045,Z 294.463,A -85,B 0,C 180,E1 -25550.234,E2 -25550.234} C_VEL
LIN {X 0,Y 123.105,Z 291.241,A -85,B 0,C 180,E1 -25560.019,E2 -25560.019} C_VEL
LIN {X 0,Y 123.834,Z 294.217,A -85,B 0,C 180,E1 -25568.176,E2 -25568.176} C_VEL
LIN {X 0,Y 127.043,Z 297.206,A -85,B 0,C 180,E1 -25576.282,E2 -25576.282} C_VEL
LIN {X 0,Y 128.07,Z 300.266,A -85,B 0,C 180,E1 -25578.826,E2 -25578.826} C_VEL
LIN {X 0,Y 130.238,Z 303.046,A -85,B 0,C 180,E1 -25582.212,E2 -25582.212} C_VEL
LIN {X 0,Y 133.077,Z 308.467,A -85,B 0,C 180,E1 -25586.691,E2 -25586.691} C_VEL
LIN {X 0,Y 133.655,Z 309.243,A -85,B 0,C 180,E1 -25587.412,E2 -25587.412} C_VEL
LIN {X 0,Y 135.64,Z 313.561,A -85,B 0,C 180,E1 -25590.196,E2 -25590.196} C_VEL
LIN {X 0,Y 138.286,Z 319.917,A -85,B 0,C 180,E1 -25594.008,E2 -25594.008} C_VEL
LIN {X 0,Y 140.245,Z 325.722,A -85,B 0,C 180,E1 -25596.985,E2 -25596.985} C_VEL
LIN {X 0,Y 141.644,Z 332.986,A -85,B 0,C 180,E1 -25600.186,E2 -25600.186} C_VEL
LIN {X 0,Y 141.994,Z 342.256,A -85,B 0,C 180,E1 -25603.882,E2 -25603.882} C_VEL
LIN {X 0,Y 141.232,Z 351.537,A -85,B 0,C 180,E1 -25607.619,E2 -25607.619} C_VEL
LIN {X 0,Y 139.87,Z 359.497,A -85,B 0,C 180,E1 -25611.092,E2 -25611.092} C_VEL
LIN {X 0,Y 138.937,Z 362.781,A -85,B 0,C 180,E1 -25612.628,E2 -25612.628} C_VEL
LIN {X 0,Y 135.574,Z 368.734,A -85,B 0,C 180,E1 -25615.235,E2 -25615.235} C_VEL
LIN {X 0,Y 131.751,Z 374.998,A -85,B 0,C 180,E1 -25618.621,E2 -25618.621} C_VEL
LIN {X 0,Y 128.387,Z 380.315,A -85,B 0,C 180,E1 -25622.271,E2 -25622.271} C_VEL
LIN {X 0,Y 124.929,Z 385.446,A -85,B 0,C 180,E1 -25626.81,E2 -25626.81} C_VEL
LIN {X 0,Y 122.237,Z 389.436,A -85,B 0,C 180,E1 -25631.566,E2 -25631.566} C_VEL
LIN {X 0,Y 120.543,Z 392.396,A -85,B 0,C 180,E1 -25636.514,E2 -25636.514} C_VEL
LIN {X 0,Y 119.355,Z 394.856,A -85,B 0,C 180,E1 -25643.237,E2 -25643.237} C_VEL
LIN {X 0,Y 119.23,Z 395.452,A -85,B 0,C 180,E1 -25646.621,E2 -25646.621} C_VEL
LIN {X 0,Y 119.324,Z 395.613,A -85,B 0,C 180,E1 -25650,E2 -25650} C_VEL
LIN {X 0,Y 119.23,Z 395.452,A -85,B 0,C 180,E1 -25653.379,E2 -25653.379} C_VEL
LIN {X 0,Y 119.347,Z 394.855,A -85,B 0,C 180,E1 -25656.763,E2 -25656.763} C_VEL
LIN {X 0,Y 120.51,Z 392.395,A -85,B 0,C 180,E1 -25663.49,E2 -25663.49} C_VEL
LIN {X 0,Y 122.237,Z 389.436,A -85,B 0,C 180,E1 -25668.434,E2 -25668.434} C_VEL
LIN {X 0,Y 124.929,Z 385.446,A -85,B 0,C 180,E1 -25673.19,E2 -25673.19} C_VEL
LIN {X 0,Y 128.395,Z 380.315,A -85,B 0,C 180,E1 -25677.727,E2 -25677.727} C_VEL
LIN {X 0,Y 131.893,Z 374.82,A -85,B 0,C 180,E1 -25681.479,E2 -25681.479} C_VEL
LIN {X 0,Y 135.538,Z 368.732,A -85,B 0,C 180,E1 -25684.776,E2 -25684.776} C_VEL
LIN {X 0,Y 138.89,Z 362.78,A -85,B 0,C 180,E1 -25687.387,E2 -25687.387} C_VEL
LIN {X 0,Y 140.226,Z 357.725,A -85,B 0,C 180,E1 -25689.717,E2 -25689.717} C_VEL
LIN {X 0,Y 141.519,Z 348.54,A -85,B 0,C 180,E1 -25693.598,E2 -25693.598} C_VEL
LIN {X 0,Y 141.967,Z 341.029,A -85,B 0,C 180,E1 -25696.597,E2 -25696.597} C_VEL
LIN {X 0,Y 141.613,Z 333.058,A -85,B 0,C 180,E1 -25699.803,E2 -25699.803} C_VEL
LIN {X 0,Y 140.252,Z 325.706,A -85,B 0,C 180,E1 -25703.017,E2 -25703.017} C_VEL
LIN {X 0,Y 137.785,Z 318.572,A -85,B 0,C 180,E1 -25706.73,E2 -25706.73} C_VEL
LIN {X 0,Y 135.641,Z 313.561,A -85,B 0,C 180,E1 -25709.803,E2 -25709.803} C_VEL
LIN {X 0,Y 133.66,Z 309.226,A -85,B 0,C 180,E1 -25712.589,E2 -25712.589} C_VEL
LIN {X 0,Y 131.895,Z 306.674,A -85,B 0,C 180,E1 -25714.934,E2 -25714.934} C_VEL
LIN {X 0,Y 130.11,Z 302.876,A -85,B 0,C 180,E1 -25717.974,E2 -25717.974} C_VEL
LIN {X 0,Y 127.601,Z 299.274,A -85,B 0,C 180,E1 -25722.141,E2 -25722.141} C_VEL
LIN {X 0,Y 126.966,Z 297.006,A -85,B 0,C 180,E1 -25723.914,E2 -25723.914} C_VEL
LIN {X 0,Y 123.062,Z 291.535,A -85,B 0,C 180,E1 -25739.367,E2 -25739.367} C_VEL
LIN {X 0,Y 123.105,Z 291.191,A -85,B 0,C 180,E1 -25739.981,E2 -25739.981} C_VEL
LIN {X 0,Y 124.117,Z 294.583,A -85,B 0,C 180,E1 -25750.05,E2 -25750.05} C_VEL
LIN {X 0,Y 124.806,Z 296.266,A -85,B 0,C 180,E1 -25752.64,E2 -25752.64} C_VEL
LIN {X 0,Y 125.463,Z 298.748,A -85,B 0,C 180,E1 -25755.09,E2 -25755.09} C_VEL
LIN {X 0,Y 127.731,Z 308.913,A -85,B 0,C 180,E1 -25762.835,E2 -25762.835} C_VEL
LIN {X 0,Y 130.3,Z 313.439,A -85,B 0,C 180,E1 -25767.266,E2 -25767.266} C_VEL
LIN {X 0,Y 132.734,Z 318.043,A -85,B 0,C 180,E1 -25771.058,E2 -25771.058} C_VEL
LIN {X 0,Y 135.192,Z 323.308,A -85,B 0,C 180,E1 -25774.855,E2 -25774.855} C_VEL
LIN {X 0,Y 137.648,Z 329.406,A -85,B 0,C 180,E1 -25778.692,E2 -25778.692} C_VEL
LIN {X 0,Y 140.042,Z 337.495,A -85,B 0,C 180,E1 -25783.291,E2 -25783.291} C_VEL
LIN {X 0,Y 141.536,Z 345.234,A -85,B 0,C 180,E1 -25787.447,E2 -25787.447} C_VEL
LIN {X 0,Y 142.347,Z 352.83,A -85,B 0,C 180,E1 -25791.55,E2 -25791.55} C_VEL
LIN {X 0,Y 142.888,Z 361.516,A -85,B 0,C 180,E1 -25796.7,E2 -25796.7} C_VEL
LIN {X 0,Y 144.42,Z 367.69,A -85,B 0,C 180,E1 -25801.117,E2 -25801.117} C_VEL
LIN {X 0,Y 146.884,Z 372.694,A -85,B 0,C 180,E1 -25805.335,E2 -25805.335} C_VEL
LIN {X 0,Y 150.26,Z 376.667,A -85,B 0,C 180,E1 -25809.247,E2 -25809.247} C_VEL
LIN {X 0,Y 154.363,Z 379.883,A -85,B 0,C 180,E1 -25812.899,E2 -25812.899} C_VEL
LIN {X 0,Y 160.959,Z 383.092,A -85,B 0,C 180,E1 -25817.39,E2 -25817.39} C_VEL
LIN {X 0,Y 170.181,Z 385.627,A -85,B 0,C 180,E1 -25822.234,E2 -25822.234} C_VEL
LIN {X 0,Y 177.694,Z 386.766,A -85,B 0,C 180,E1 -25825.463,E2 -25825.463} C_VEL
LIN {X 0,Y 183.869,Z 387.166,A -85,B 0,C 180,E1 -25827.81,E2 -25827.81} C_VEL
LIN {X 0,Y 189.96,Z 387.159,A -85,B 0,C 180,E1 -25830,E2 -25830} C_VEL
LIN {X 0,Y 182.859,Z 387.104,A -85,B 0,C 180,E1 -25832.565,E2 -25832.565} C_VEL
LIN {X 0,Y 176.344,Z 386.625,A -85,B 0,C 180,E1 -25835.092,E2 -25835.092} C_VEL
LIN {X 0,Y 166.145,Z 384.706,A -85,B 0,C 180,E1 -25839.741,E2 -25839.741} C_VEL
LIN {X 0,Y 159.11,Z 382.335,A -85,B 0,C 180,E1 -25843.728,E2 -25843.728} C_VEL
LIN {X 0,Y 154.356,Z 379.891,A -85,B 0,C 180,E1 -25847.094,E2 -25847.094} C_VEL
LIN {X 0,Y 148.862,Z 375.325,A -85,B 0,C 180,E1 -25852.19,E2 -25852.19} C_VEL
LIN {X 0,Y 145.16,Z 369.586,A -85,B 0,C 180,E1 -25857.381,E2 -25857.381} C_VEL
LIN {X 0,Y 143.24,Z 363.714,A -85,B 0,C 180,E1 -25861.832,E2 -25861.832} C_VEL
LIN {X 0,Y 142.545,Z 358.191,A -85,B 0,C 180,E1 -25865.401,E2 -25865.401} C_VEL
LIN {X 0,Y 142.245,Z 351.388,A -85,B 0,C 180,E1 -25869.216,E2 -25869.216} C_VEL
LIN {X 0,Y 141.336,Z 344.124,A -85,B 0,C 180,E1 -25873.14,E2 -25873.14} C_VEL
LIN {X 0,Y 139.764,Z 336.48,A -85,B 0,C 180,E1 -25877.273,E2 -25877.273} C_VEL
LIN {X 0,Y 137.647,Z 329.408,A -85,B 0,C 180,E1 -25881.308,E2 -25881.308} C_VEL
LIN {X 0,Y 134.599,Z 321.965,A -85,B 0,C 180,E1 -25886.081,E2 -25886.081} C_VEL
LIN {X 0,Y 132.288,Z 316.892,A -85,B 0,C 180,E1 -25889.711,E2 -25889.711} C_VEL
LIN {X 0,Y 129.361,Z 311.928,A -85,B 0,C 180,E1 -25894.26,E2 -25894.26} C_VEL
LIN {X 0,Y 127.64,Z 308.701,A -85,B 0,C 180,E1 -25897.351,E2 -25897.351} C_VEL
LIN {X 0,Y 125.096,Z 305.5,A -85,B 0,C 180,E1 -25902.024,E2 -25902.024} C_VEL
LIN {X 0,Y 124.568,Z 304.037,A -85,B 0,C 180,E1 -25903.635,E2 -25903.635} C_VEL
LIN {X 0,Y 122.116,Z 301.125,A -85,B 0,C 180,E1 -25910.914,E2 -25910.914} C_VEL
LIN {X 0,Y 121.403,Z 298.413,A -85,B 0,C 180,E1 -25920.227,E2 -25920.227} C_VEL
LIN {X 0,Y 124.426,Z 303.442,A -85,B 0,C 180,E1 -25934.743,E2 -25934.743} C_VEL
LIN {X 0,Y 125.286,Z 306.176,A -85,B 0,C 180,E1 -25937.522,E2 -25937.522} C_VEL
LIN {X 0,Y 127.077,Z 309.046,A -85,B 0,C 180,E1 -25941.087,E2 -25941.087} C_VEL
LIN {X 0,Y 130.146,Z 315.119,A -85,B 0,C 180,E1 -25946.474,E2 -25946.474} C_VEL
LIN {X 0,Y 132.745,Z 321.885,A -85,B 0,C 180,E1 -25951.096,E2 -25951.096} C_VEL
LIN {X 0,Y 134.325,Z 326.45,A -85,B 0,C 180,E1 -25953.898,E2 -25953.898} C_VEL
LIN {X 0,Y 135.672,Z 331.828,A -85,B 0,C 180,E1 -25956.765,E2 -25956.765} C_VEL
LIN {X 0,Y 136.247,Z 337.232,A -85,B 0,C 180,E1 -25959.311,E2 -25959.311} C_VEL
LIN {X 0,Y 136.161,Z 345.051,A -85,B 0,C 180,E1 -25962.69,E2 -25962.69} C_VEL
LIN {X 0,Y 135.391,Z 351.681,A -85,B 0,C 180,E1 -25965.515,E2 -25965.515} C_VEL
LIN {X 0,Y 133.973,Z 359.286,A -85,B 0,C 180,E1 -25969.026,E2 -25969.026} C_VEL
LIN {X 0,Y 132.446,Z 364.214,A -85,B 0,C 180,E1 -25971.429,E2 -25971.429} C_VEL
LIN {X 0,Y 127.265,Z 372.543,A -85,B 0,C 180,E1 -25975.527,E2 -25975.527} C_VEL
LIN {X 0,Y 123.538,Z 378.204,A -85,B 0,C 180,E1 -25979.203,E2 -25979.203} C_VEL
LIN {X 0,Y 119.56,Z 383.696,A -85,B 0,C 180,E1 -25983.841,E2 -25983.841} C_VEL
LIN {X 0,Y 116.348,Z 388.022,A -85,B 0,C 180,E1 -25988.751,E2 -25988.751} C_VEL
LIN {X 0,Y 114.759,Z 390.393,A -85,B 0,C 180,E1 -25992.17,E2 -25992.17} C_VEL
LIN {X 0,Y 113.631,Z 392.2,A -85,B 0,C 180,E1 -25995.677,E2 -25995.677} C_VEL
LIN {X 0,Y 112.292,Z 394.66,A -85,B 0,C 180,E1 -26002.809,E2 -26002.809} C_VEL
LIN {X 0,Y 112.146,Z 395.258,A -85,B 0,C 180,E1 -26006.407,E2 -26006.407} C_VEL
LIN {X 0,Y 112.237,Z 395.418,A -85,B 0,C 180,E1 -26010,E2 -26010} C_VEL
LIN {X 0,Y 112.145,Z 395.258,A -85,B 0,C 180,E1 -26013.593,E2 -26013.593} C_VEL
LIN {X 0,Y 112.283,Z 394.66,A -85,B 0,C 180,E1 -26017.191,E2 -26017.191} C_VEL
LIN {X 0,Y 113.589,Z 392.199,A -85,B 0,C 180,E1 -26024.329,E2 -26024.329} C_VEL
LIN {X 0,Y 115.493,Z 389.241,A -85,B 0,C 180,E1 -26029.553,E2 -26029.553} C_VEL
LIN {X 0,Y 118.42,Z 385.25,A -85,B 0,C 180,E1 -26034.546,E2 -26034.546} C_VEL
LIN {X 0,Y 122.147,Z 380.121,A -85,B 0,C 180,E1 -26039.279,E2 -26039.279} C_VEL
LIN {X 0,Y 125.486,Z 375.189,A -85,B 0,C 180,E1 -26042.821,E2 -26042.821} C_VEL
LIN {X 0,Y 129.745,Z 368.537,A -85,B 0,C 180,E1 -26046.572,E2 -26046.572} C_VEL
LIN {X 0,Y 132.427,Z 364.213,A -85,B 0,C 180,E1 -26048.577,E2 -26048.577} C_VEL
LIN {X 0,Y 133.977,Z 359.286,A -85,B 0,C 180,E1 -26050.972,E2 -26050.972} C_VEL
LIN {X 0,Y 135.728,Z 349.579,A -85,B 0,C 180,E1 -26055.393,E2 -26055.393} C_VEL
LIN {X 0,Y 136.285,Z 341.559,A -85,B 0,C 180,E1 -26058.872,E2 -26058.872} C_VEL
LIN {X 0,Y 136.062,Z 335.143,A -85,B 0,C 180,E1 -26061.677,E2 -26061.677} C_VEL
LIN {X 0,Y 135.301,Z 330.009,A -85,B 0,C 180,E1 -26064.129,E2 -26064.129} C_VEL
LIN {X 0,Y 133.236,Z 323.074,A -85,B 0,C 180,E1 -26068.146,E2 -26068.146} C_VEL
LIN {X 0,Y 131.357,Z 318.454,A -85,B 0,C 180,E1 -26071.196,E2 -26071.196} C_VEL
LIN {X 0,Y 130.155,Z 315.096,A -85,B 0,C 180,E1 -26073.528,E2 -26073.528} C_VEL
LIN {X 0,Y 127.085,Z 309.021,A -85,B 0,C 180,E1 -26078.915,E2 -26078.915} C_VEL
LIN {X 0,Y 124.914,Z 304.978,A -85,B 0,C 180,E1 -26083.643,E2 -26083.643} C_VEL
LIN {X 0,Y 124.433,Z 303.416,A -85,B 0,C 180,E1 -26085.258,E2 -26085.258} C_VEL
LIN {X 0,Y 121.42,Z 298.331,A -85,B 0,C 180,E1 -26099.981,E2 -26099.981} C_VEL
LIN {X 0,Y 123.316,Z 302.598,A -85,B 0,C 180,E1 -26113.157,E2 -26113.157} C_VEL
LIN {X 0,Y 124.611,Z 304.171,A -85,B 0,C 180,E1 -26116.51,E2 -26116.51} C_VEL
LIN {X 0,Y 125.825,Z 306.647,A -85,B 0,C 180,E1 -26119.559,E2 -26119.559} C_VEL
LIN {X 0,Y 127.731,Z 308.913,A -85,B 0,C 180,E1 -26122.835,E2 -26122.835} C_VEL
LIN {X 0,Y 128.591,Z 312.082,A -85,B 0,C 180,E1 -26125.045,E2 -26125.045} C_VEL
LIN {X 0,Y 129.212,Z 318.423,A -85,B 0,C 180,E1 -26128.435,E2 -26128.435} C_VEL
LIN {X 0,Y 129.916,Z 326.088,A -85,B 0,C 180,E1 -26132.512,E2 -26132.512} C_VEL
LIN {X 0,Y 130.585,Z 328.274,A -85,B 0,C 180,E1 -26133.95,E2 -26133.95} C_VEL
LIN {X 0,Y 132.649,Z 334.359,A -85,B 0,C 180,E1 -26138.172,E2 -26138.172} C_VEL
LIN {X 0,Y 134.223,Z 340.607,A -85,B 0,C 180,E1 -26142.059,E2 -26142.059} C_VEL
LIN {X 0,Y 135.294,Z 346.529,A -85,B 0,C 180,E1 -26145.553,E2 -26145.553} C_VEL
LIN {X 0,Y 135.936,Z 353.661,A -85,B 0,C 180,E1 -26149.736,E2 -26149.736} C_VEL
LIN {X 0,Y 136.069,Z 361.274,A -85,B 0,C 180,E1 -26154.476,E2 -26154.476} C_VEL
LIN {X 0,Y 136.962,Z 367.594,A -85,B 0,C 180,E1 -26159.128,E2 -26159.128} C_VEL
LIN {X 0,Y 139.179,Z 373.214,A -85,B 0,C 180,E1 -26164.117,E2 -26164.117} C_VEL
LIN {X 0,Y 141.938,Z 376.938,A -85,B 0,C 180,E1 -26167.995,E2 -26167.995} C_VEL
LIN {X 0,Y 146.925,Z 380.932,A -85,B 0,C 180,E1 -26173.007,E2 -26173.007} C_VEL
LIN {X 0,Y 151.751,Z 383.351,A -85,B 0,C 180,E1 -26176.611,E2 -26176.611} C_VEL
LIN {X 0,Y 157.025,Z 385.061,A -85,B 0,C 180,E1 -26179.846,E2 -26179.846} C_VEL
LIN {X 0,Y 168.011,Z 387.028,A -85,B 0,C 180,E1 -26185.201,E2 -26185.201} C_VEL
LIN {X 0,Y 175.728,Z 387.499,A -85,B 0,C 180,E1 -26188.268,E2 -26188.268} C_VEL
LIN {X 0,Y 180.49,Z 387.414,A -85,B 0,C 180,E1 -26190,E2 -26190} C_VEL
LIN {X 0,Y 174.223,Z 387.429,A -85,B 0,C 180,E1 -26192.312,E2 -26192.312} C_VEL
LIN {X 0,Y 168.012,Z 387.028,A -85,B 0,C 180,E1 -26194.799,E2 -26194.799} C_VEL
LIN {X 0,Y 156.69,Z 384.964,A -85,B 0,C 180,E1 -26200.335,E2 -26200.335} C_VEL
LIN {X 0,Y 149.428,Z 382.303,A -85,B 0,C 180,E1 -26204.99,E2 -26204.99} C_VEL
LIN {X 0,Y 145.418,Z 380.027,A -85,B 0,C 180,E1 -26208.315,E2 -26208.315} C_VEL
LIN {X 0,Y 140.707,Z 375.568,A -85,B 0,C 180,E1 -26213.552,E2 -26213.552} C_VEL
LIN {X 0,Y 137.608,Z 369.844,A -85,B 0,C 180,E1 -26219.004,E2 -26219.004} C_VEL
LIN {X 0,Y 136.262,Z 363.963,A -85,B 0,C 180,E1 -26223.657,E2 -26223.657} C_VEL
LIN {X 0,Y 136.028,Z 358.411,A -85,B 0,C 180,E1 -26227.377,E2 -26227.377} C_VEL
LIN {X 0,Y 135.817,Z 351.971,A -85,B 0,C 180,E1 -26231.28,E2 -26231.28} C_VEL
LIN {X 0,Y 135.035,Z 344.993,A -85,B 0,C 180,E1 -26235.392,E2 -26235.392} C_VEL
LIN {X 0,Y 133.501,Z 337.425,A -85,B 0,C 180,E1 -26239.946,E2 -26239.946} C_VEL
LIN {X 0,Y 131.578,Z 331.078,A -85,B 0,C 180,E1 -26244.042,E2 -26244.042} C_VEL
LIN {X 0,Y 129.446,Z 325.567,A -85,B 0,C 180,E1 -26248.062,E2 -26248.062} C_VEL
LIN {X 0,Y 128.245,Z 322.492,A -85,B 0,C 180,E1 -26250.471,E2 -26250.471} C_VEL
LIN {X 0,Y 126.553,Z 319.08,A -85,B 0,C 180,E1 -26253.646,E2 -26253.646} C_VEL
LIN {X 0,Y 124.189,Z 314.564,A -85,B 0,C 180,E1 -26258.439,E2 -26258.439} C_VEL
LIN {X 0,Y 122.151,Z 311.36,A -85,B 0,C 180,E1 -26263.302,E2 -26263.302} C_VEL
LIN {X 0,Y 121.036,Z 309.459,A -85,B 0,C 180,E1 -26266.591,E2 -26266.591} C_VEL
LIN {X 0,Y 119.426,Z 305.28,A -85,B 0,C 180,E1 -26280.02,E2 -26280.02} C_VEL
LIN {X 0,Y 121.484,Z 309.708,A -85,B 0,C 180,E1 -26293.399,E2 -26293.399} C_VEL
LIN {X 0,Y 121.999,Z 310.857,A -85,B 0,C 180,E1 -26295.044,E2 -26295.044} C_VEL
LIN {X 0,Y 122.923,Z 313.375,A -85,B 0,C 180,E1 -26297.87,E2 -26297.87} C_VEL
LIN {X 0,Y 124.478,Z 316.432,A -85,B 0,C 180,E1 -26301.549,E2 -26301.549} C_VEL
LIN {X 0,Y 126.334,Z 320.808,A -85,B 0,C 180,E1 -26305.559,E2 -26305.559} C_VEL
LIN {X 0,Y 128.509,Z 327.407,A -85,B 0,C 180,E1 -26310.408,E2 -26310.408} C_VEL
LIN {X 0,Y 130.259,Z 333.997,A -85,B 0,C 180,E1 -26314.537,E2 -26314.537} C_VEL
LIN {X 0,Y 130.743,Z 339.057,A -85,B 0,C 180,E1 -26317.23,E2 -26317.23} C_VEL
LIN {X 0,Y 130.565,Z 345.4,A -85,B 0,C 180,E1 -26320.256,E2 -26320.256} C_VEL
LIN {X 0,Y 129.842,Z 351.459,A -85,B 0,C 180,E1 -26323.055,E2 -26323.055} C_VEL
LIN {X 0,Y 128.2,Z 359.318,A -85,B 0,C 180,E1 -26326.904,E2 -26326.904} C_VEL
LIN {X 0,Y 126.79,Z 364.013,A -85,B 0,C 180,E1 -26329.361,E2 -26329.361} C_VEL
LIN {X 0,Y 124.137,Z 368.343,A -85,B 0,C 180,E1 -26331.483,E2 -26331.483} C_VEL
LIN {X 0,Y 119.785,Z 374.637,A -85,B 0,C 180,E1 -26335.088,E2 -26335.088} C_VEL
LIN {X 0,Y 115.975,Z 379.925,A -85,B 0,C 180,E1 -26338.997,E2 -26338.997} C_VEL
LIN {X 0,Y 111.983,Z 385.055,A -85,B 0,C 180,E1 -26343.94,E2 -26343.94} C_VEL
LIN {X 0,Y 108.807,Z 389.045,A -85,B 0,C 180,E1 -26349.192,E2 -26349.192} C_VEL
LIN {X 0,Y 106.717,Z 392.004,A -85,B 0,C 180,E1 -26354.727,E2 -26354.727} C_VEL
LIN {X 0,Y 105.251,Z 394.466,A -85,B 0,C 180,E1 -26362.326,E2 -26362.326} C_VEL
LIN {X 0,Y 105.059,Z 395.063,A -85,B 0,C 180,E1 -26366.164,E2 -26366.164} C_VEL
LIN {X 0,Y 105.142,Z 395.224,A -85,B 0,C 180,E1 -26370,E2 -26370} C_VEL
LIN {X 0,Y 105.058,Z 395.063,A -85,B 0,C 180,E1 -26373.836,E2 -26373.836} C_VEL
LIN {X 0,Y 105.242,Z 394.466,A -85,B 0,C 180,E1 -26377.675,E2 -26377.675} C_VEL
LIN {X 0,Y 106.68,Z 392.003,A -85,B 0,C 180,E1 -26385.278,E2 -26385.278} C_VEL
LIN {X 0,Y 108.807,Z 389.045,A -85,B 0,C 180,E1 -26390.808,E2 -26390.808} C_VEL
LIN {X 0,Y 111.983,Z 385.055,A -85,B 0,C 180,E1 -26396.059,E2 -26396.059} C_VEL
LIN {X 0,Y 115.993,Z 379.926,A -85,B 0,C 180,E1 -26400.997,E2 -26400.997} C_VEL
LIN {X 0,Y 119.879,Z 374.524,A -85,B 0,C 180,E1 -26404.981,E2 -26404.981} C_VEL
LIN {X 0,Y 124.095,Z 368.341,A -85,B 0,C 180,E1 -26408.533,E2 -26408.533} C_VEL
LIN {X 0,Y 126.792,Z 364.013,A -85,B 0,C 180,E1 -26410.638,E2 -26410.638} C_VEL
LIN {X 0,Y 128.684,Z 357.342,A -85,B 0,C 180,E1 -26414.109,E2 -26414.109} C_VEL
LIN {X 0,Y 130.175,Z 349.355,A -85,B 0,C 180,E1 -26417.93,E2 -26417.93} C_VEL
LIN {X 0,Y 130.82,Z 341.04,A -85,B 0,C 180,E1 -26421.824,E2 -26421.824} C_VEL
LIN {X 0,Y 130.459,Z 335.558,A -85,B 0,C 180,E1 -26424.582,E2 -26424.582} C_VEL
LIN {X 0,Y 129.262,Z 329.822,A -85,B 0,C 180,E1 -26427.968,E2 -26427.968} C_VEL
LIN {X 0,Y 127.526,Z 324.281,A -85,B 0,C 180,E1 -26431.853,E2 -26431.853} C_VEL
LIN {X 0,Y 125.914,Z 319.932,A -85,B 0,C 180,E1 -26435.234,E2 -26435.234} C_VEL
LIN {X 0,Y 123.811,Z 314.922,A -85,B 0,C 180,E1 -26440.069,E2 -26440.069} C_VEL
LIN {X 0,Y 122.012,Z 310.816,A -85,B 0,C 180,E1 -26444.958,E2 -26444.958} C_VEL
LIN {X 0,Y 121.481,Z 309.718,A -85,B 0,C 180,E1 -26446.601,E2 -26446.601} C_VEL
LIN {X 0,Y 119.422,Z 305.292,A -85,B 0,C 180,E1 -26459.98,E2 -26459.98} C_VEL
LIN {X 0,Y 121.033,Z 309.465,A -85,B 0,C 180,E1 -26473.41,E2 -26473.41} C_VEL
LIN {X 0,Y 122.698,Z 312.549,A -85,B 0,C 180,E1 -26478.342,E2 -26478.342} C_VEL
LIN {X 0,Y 124.31,Z 314.898,A -85,B 0,C 180,E1 -26481.893,E2 -26481.893} C_VEL
LIN {X 0,Y 126.536,Z 319.125,A -85,B 0,C 180,E1 -26486.358,E2 -26486.358} C_VEL
LIN {X 0,Y 128.591,Z 323.578,A -85,B 0,C 180,E1 -26490.344,E2 -26490.344} C_VEL
LIN {X 0,Y 130.585,Z 328.274,A -85,B 0,C 180,E1 -26493.95,E2 -26493.95} C_VEL
LIN {X 0,Y 131.269,Z 331.77,A -85,B 0,C 180,E1 -26496.015,E2 -26496.015} C_VEL
LIN {X 0,Y 131.047,Z 335.856,A -85,B 0,C 180,E1 -26497.915,E2 -26497.915} C_VEL
LIN {X 0,Y 129.553,Z 344.389,A -85,B 0,C 180,E1 -26501.654,E2 -26501.654} C_VEL
LIN {X 0,Y 129.189,Z 348.2,A -85,B 0,C 180,E1 -26503.702,E2 -26503.702} C_VEL
LIN {X 0,Y 129.246,Z 349.346,A -85,B 0,C 180,E1 -26504.423,E2 -26504.423} C_VEL
LIN {X 0,Y 129.61,Z 355.684,A -85,B 0,C 180,E1 -26508.513,E2 -26508.513} C_VEL
LIN {X 0,Y 129.495,Z 361.499,A -85,B 0,C 180,E1 -26512.371,E2 -26512.371} C_VEL
LIN {X 0,Y 129.832,Z 367.824,A -85,B 0,C 180,E1 -26517.228,E2 -26517.228} C_VEL
LIN {X 0,Y 131.746,Z 373.97,A -85,B 0,C 180,E1 -26523.027,E2 -26523.027} C_VEL
LIN {X 0,Y 133.912,Z 377.379,A -85,B 0,C 180,E1 -26526.821,E2 -26526.821} C_VEL
LIN {X 0,Y 138.597,Z 381.429,A -85,B 0,C 180,E1 -26532.287,E2 -26532.287} C_VEL
LIN {X 0,Y 144.242,Z 384.193,A -85,B 0,C 180,E1 -26536.939,E2 -26536.939} C_VEL
LIN {X 0,Y 152.604,Z 386.418,A -85,B 0,C 180,E1 -26542.059,E2 -26542.059} C_VEL
LIN {X 0,Y 161.897,Z 387.529,A -85,B 0,C 180,E1 -26546.487,E2 -26546.487} C_VEL
LIN {X 0,Y 170.888,Z 387.672,A -85,B 0,C 180,E1 -26550,E2 -26550} C_VEL
LIN {X 0,Y 161.897,Z 387.528,A -85,B 0,C 180,E1 -26553.514,E2 -26553.514} C_VEL
LIN {X 0,Y 152.589,Z 386.419,A -85,B 0,C 180,E1 -26557.942,E2 -26557.942} C_VEL
LIN {X 0,Y 144.235,Z 384.201,A -85,B 0,C 180,E1 -26563.049,E2 -26563.049} C_VEL
LIN {X 0,Y 136.993,Z 380.375,A -85,B 0,C 180,E1 -26569.363,E2 -26569.363} C_VEL
LIN {X 0,Y 132.424,Z 375.293,A -85,B 0,C 180,E1 -26575.597,E2 -26575.597} C_VEL
LIN {X 0,Y 130.406,Z 370.456,A -85,B 0,C 180,E1 -26580.467,E2 -26580.467} C_VEL
LIN {X 0,Y 129.52,Z 364.345,A -85,B 0,C 180,E1 -26585.555,E2 -26585.555} C_VEL
LIN {X 0,Y 129.622,Z 358.359,A -85,B 0,C 180,E1 -26589.749,E2 -26589.749} C_VEL
LIN {X 0,Y 129.471,Z 352.169,A -85,B 0,C 180,E1 -26593.816,E2 -26593.816} C_VEL
LIN {X 0,Y 128.86,Z 346.082,A -85,B 0,C 180,E1 -26597.758,E2 -26597.758} C_VEL
LIN {X 0,Y 127.437,Z 338.777,A -85,B 0,C 180,E1 -26602.679,E2 -26602.679} C_VEL
LIN {X 0,Y 125.351,Z 331.964,A -85,B 0,C 180,E1 -26607.839,E2 -26607.839} C_VEL
LIN {X 0,Y 124.006,Z 327.965,A -85,B 0,C 180,E1 -26611.218,E2 -26611.218} C_VEL
LIN {X 0,Y 122.505,Z 324.598,A -85,B 0,C 180,E1 -26614.538,E2 -26614.538} C_VEL
LIN {X 0,Y 120.592,Z 320.373,A -85,B 0,C 180,E1 -26619.555,E2 -26619.555} C_VEL
LIN {X 0,Y 118.327,Z 316.305,A -85,B 0,C 180,E1 -26626.278,E2 -26626.278} C_VEL
LIN {X 0,Y 116.976,Z 313.98,A -85,B 0,C 180,E1 -26633.119,E2 -26633.119} C_VEL
LIN {X 0,Y 117.09,Z 312.086,A -85,B 0,C 180,E1 -26640.02,E2 -26640.02} C_VEL
LIN {X 0,Y 117.9,Z 315.267,A -85,B 0,C 180,E1 -26650.321,E2 -26650.321} C_VEL
LIN {X 0,Y 118.838,Z 316.688,A -85,B 0,C 180,E1 -26653.703,E2 -26653.703} C_VEL
LIN {X 0,Y 120.875,Z 322.082,A -85,B 0,C 180,E1 -26660.437,E2 -26660.437} C_VEL
LIN {X 0,Y 122.017,Z 325.47,A -85,B 0,C 180,E1 -26663.797,E2 -26663.797} C_VEL
LIN {X 0,Y 123.904,Z 331.978,A -85,B 0,C 180,E1 -26669.072,E2 -26669.072} C_VEL
LIN {X 0,Y 125.094,Z 337.949,A -85,B 0,C 180,E1 -26673.234,E2 -26673.234} C_VEL
LIN {X 0,Y 125.388,Z 342.53,A -85,B 0,C 180,E1 -26675.846,E2 -26675.846} C_VEL
LIN {X 0,Y 124.757,Z 349.674,A -85,B 0,C 180,E1 -26679.537,E2 -26679.537} C_VEL
LIN {X 0,Y 122.825,Z 358.456,A -85,B 0,C 180,E1 -26684.05,E2 -26684.05} C_VEL
LIN {X 0,Y 120.548,Z 365.385,A -85,B 0,C 180,E1 -26687.899,E2 -26687.899} C_VEL
LIN {X 0,Y 114.867,Z 373.308,A -85,B 0,C 180,E1 -26692.279,E2 -26692.279} C_VEL
LIN {X 0,Y 109.929,Z 379.73,A -85,B 0,C 180,E1 -26697.084,E2 -26697.084} C_VEL
LIN {X 0,Y 105.615,Z 384.859,A -85,B 0,C 180,E1 -26702.239,E2 -26702.239} C_VEL
LIN {X 0,Y 102.188,Z 388.85,A -85,B 0,C 180,E1 -26707.774,E2 -26707.774} C_VEL
LIN {X 0,Y 99.841,Z 391.808,A -85,B 0,C 180,E1 -26713.647,E2 -26713.647} C_VEL
LIN {X 0,Y 98.209,Z 394.271,A -85,B 0,C 180,E1 -26721.772,E2 -26721.772} C_VEL
LIN {X 0,Y 97.968,Z 394.868,A -85,B 0,C 180,E1 -26725.886,E2 -26725.886} C_VEL
LIN {X 0,Y 98.04,Z 395.029,A -85,B 0,C 180,E1 -26730,E2 -26730} C_VEL
LIN {X 0,Y 97.967,Z 394.868,A -85,B 0,C 180,E1 -26734.114,E2 -26734.114} C_VEL
LIN {X 0,Y 98.179,Z 394.27,A -85,B 0,C 180,E1 -26738.231,E2 -26738.231} C_VEL
LIN {X 0,Y 99.811,Z 391.808,A -85,B 0,C 180,E1 -26746.358,E2 -26746.358} C_VEL
LIN {X 0,Y 102.188,Z 388.85,A -85,B 0,C 180,E1 -26752.226,E2 -26752.226} C_VEL
LIN {X 0,Y 105.616,Z 384.859,A -85,B 0,C 180,E1 -26757.761,E2 -26757.761} C_VEL
LIN {X 0,Y 109.954,Z 379.73,A -85,B 0,C 180,E1 -26762.908,E2 -26762.908} C_VEL
LIN {X 0,Y 114.863,Z 373.308,A -85,B 0,C 180,E1 -26767.723,E2 -26767.723} C_VEL
LIN {X 0,Y 120.539,Z 365.385,A -85,B 0,C 180,E1 -26772.105,E2 -26772.105} C_VEL
LIN {X 0,Y 122.831,Z 358.42,A -85,B 0,C 180,E1 -26775.971,E2 -26775.971} C_VEL
LIN {X 0,Y 124.584,Z 350.715,A -85,B 0,C 180,E1 -26779.934,E2 -26779.934} C_VEL
LIN {X 0,Y 125.308,Z 343.606,A -85,B 0,C 180,E1 -26783.573,E2 -26783.573} C_VEL
LIN {X 0,Y 125.093,Z 337.95,A -85,B 0,C 180,E1 -26786.765,E2 -26786.765} C_VEL
LIN {X 0,Y 123.9,Z 331.938,A -85,B 0,C 180,E1 -26790.952,E2 -26790.952} C_VEL
LIN {X 0,Y 122.007,Z 325.491,A -85,B 0,C 180,E1 -26796.201,E2 -26796.201} C_VEL
LIN {X 0,Y 120.89,Z 322.045,A -85,B 0,C 180,E1 -26799.566,E2 -26799.566} C_VEL
LIN {X 0,Y 118.848,Z 316.665,A -85,B 0,C 180,E1 -26806.298,E2 -26806.298} C_VEL
LIN {X 0,Y 117.207,Z 314.24,A -85,B 0,C 180,E1 -26813.092,E2 -26813.092} C_VEL
LIN {X 0,Y 117.091,Z 312.085,A -85,B 0,C 180,E1 -26819.98,E2 -26819.98} C_VEL
LIN {X 0,Y 117.495,Z 315.018,A -85,B 0,C 180,E1 -26830.316,E2 -26830.316} C_VEL
LIN {X 0,Y 118.325,Z 316.308,A -85,B 0,C 180,E1 -26833.723,E2 -26833.723} C_VEL
LIN {X 0,Y 120.58,Z 320.4,A -85,B 0,C 180,E1 -26840.448,E2 -26840.448} C_VEL
LIN {X 0,Y 122.487,Z 324.635,A -85,B 0,C 180,E1 -26845.466,E2 -26845.466} C_VEL
LIN {X 0,Y 124.324,Z 329.035,A -85,B 0,C 180,E1 -26849.625,E2 -26849.625} C_VEL
LIN {X 0,Y 126.418,Z 335.194,A -85,B 0,C 180,E1 -26854.713,E2 -26854.713} C_VEL
LIN {X 0,Y 127.788,Z 340.556,A -85,B 0,C 180,E1 -26858.569,E2 -26858.569} C_VEL
LIN {X 0,Y 128.874,Z 346.068,A -85,B 0,C 180,E1 -26862.24,E2 -26862.24} C_VEL
LIN {X 0,Y 129.246,Z 349.346,A -85,B 0,C 180,E1 -26864.423,E2 -26864.423} C_VEL
LIN {X 0,Y 129.138,Z 351.807,A -85,B 0,C 180,E1 -26865.823,E2 -26865.823} C_VEL
LIN {X 0,Y 128.489,Z 354.344,A -85,B 0,C 180,E1 -26867.14,E2 -26867.14} C_VEL
LIN {X 0,Y 126.265,Z 359.564,A -85,B 0,C 180,E1 -26869.696,E2 -26869.696} C_VEL
LIN {X 0,Y 123.513,Z 365.505,A -85,B 0,C 180,E1 -26873.152,E2 -26873.152} C_VEL
LIN {X 0,Y 122.991,Z 368.463,A -85,B 0,C 180,E1 -26875.52,E2 -26875.52} C_VEL
LIN {X 0,Y 123.599,Z 372.384,A -85,B 0,C 180,E1 -26879.22,E2 -26879.22} C_VEL
LIN {X 0,Y 126.046,Z 377.821,A -85,B 0,C 180,E1 -26885.522,E2 -26885.522} C_VEL
LIN {X 0,Y 130.037,Z 381.676,A -85,B 0,C 180,E1 -26891.079,E2 -26891.079} C_VEL
LIN {X 0,Y 133.68,Z 383.862,A -85,B 0,C 180,E1 -26894.76,E2 -26894.76} C_VEL
LIN {X 0,Y 142.265,Z 386.506,A -85,B 0,C 180,E1 -26900.991,E2 -26900.991} C_VEL
LIN {X 0,Y 148.749,Z 387.55,A -85,B 0,C 180,E1 -26904.578,E2 -26904.578} C_VEL
LIN {X 0,Y 154.771,Z 387.957,A -85,B 0,C 180,E1 -26907.397,E2 -26907.397} C_VEL
LIN {X 0,Y 161.25,Z 387.932,A -85,B 0,C 180,E1 -26910,E2 -26910} C_VEL
LIN {X 0,Y 154.729,Z 387.951,A -85,B 0,C 180,E1 -26912.636,E2 -26912.636} C_VEL
LIN {X 0,Y 148.259,Z 387.518,A -85,B 0,C 180,E1 -26915.654,E2 -26915.654} C_VEL
LIN {X 0,Y 138.038,Z 385.477,A -85,B 0,C 180,E1 -26921.75,E2 -26921.75} C_VEL
LIN {X 0,Y 132.056,Z 382.997,A -85,B 0,C 180,E1 -26926.746,E2 -26926.746} C_VEL
LIN {X 0,Y 127.061,Z 379.085,A -85,B 0,C 180,E1 -26932.779,E2 -26932.779} C_VEL
LIN {X 0,Y 124.982,Z 376.044,A -85,B 0,C 180,E1 -26936.734,E2 -26936.734} C_VEL
LIN {X 0,Y 123.159,Z 370.281,A -85,B 0,C 180,E1 -26942.825,E2 -26942.825} C_VEL
LIN {X 0,Y 122.983,Z 364.379,A -85,B 0,C 180,E1 -26947.91,E2 -26947.91} C_VEL
LIN {X 0,Y 123.36,Z 358.537,A -85,B 0,C 180,E1 -26952.247,E2 -26952.247} C_VEL
LIN {X 0,Y 123.205,Z 352.18,A -85,B 0,C 180,E1 -26956.832,E2 -26956.832} C_VEL
LIN {X 0,Y 122.457,Z 345.18,A -85,B 0,C 180,E1 -26961.934,E2 -26961.934} C_VEL
LIN {X 0,Y 121.161,Z 338.983,A -85,B 0,C 180,E1 -26966.83,E2 -26966.83} C_VEL
LIN {X 0,Y 119.498,Z 333.247,A -85,B 0,C 180,E1 -26971.957,E2 -26971.957} C_VEL
LIN {X 0,Y 118.355,Z 330.053,A -85,B 0,C 180,E1 -26975.462,E2 -26975.462} C_VEL
LIN {X 0,Y 116.637,Z 325.994,A -85,B 0,C 180,E1 -26980.669,E2 -26980.669} C_VEL
LIN {X 0,Y 115.305,Z 322.992,A -85,B 0,C 180,E1 -26985.911,E2 -26985.911} C_VEL
LIN {X 0,Y 114.124,Z 320.556,A -85,B 0,C 180,E1 -26992.946,E2 -26992.946} C_VEL
LIN {X 0,Y 114.247,Z 318.684,A -85,B 0,C 180,E1 -27000.021,E2 -27000.021} C_VEL
LIN {X 0,Y 115.046,Z 321.901,A -85,B 0,C 180,E1 -27010.58,E2 -27010.58} C_VEL
LIN {X 0,Y 115.741,Z 323.738,A -85,B 0,C 180,E1 -27014.077,E2 -27014.077} C_VEL
LIN {X 0,Y 116.945,Z 327.562,A -85,B 0,C 180,E1 -27019.321,E2 -27019.321} C_VEL
LIN {X 0,Y 117.887,Z 330.834,A -85,B 0,C 180,E1 -27022.774,E2 -27022.774} C_VEL
LIN {X 0,Y 119.2,Z 336.916,A -85,B 0,C 180,E1 -27028.164,E2 -27028.164} C_VEL
LIN {X 0,Y 119.979,Z 341.869,A -85,B 0,C 180,E1 -27031.837,E2 -27031.837} C_VEL
LIN {X 0,Y 119.875,Z 346.579,A -85,B 0,C 180,E1 -27034.838,E2 -27034.838} C_VEL
LIN {X 0,Y 118.686,Z 353.57,A -85,B 0,C 180,E1 -27038.74,E2 -27038.74} C_VEL
LIN {X 0,Y 116.662,Z 360.691,A -85,B 0,C 180,E1 -27042.747,E2 -27042.747} C_VEL
LIN {X 0,Y 115.084,Z 365.179,A -85,B 0,C 180,E1 -27045.391,E2 -27045.391} C_VEL
LIN {X 0,Y 114.351,Z 366.575,A -85,B 0,C 180,E1 -27046.258,E2 -27046.258} C_VEL
LIN {X 0,Y 109.314,Z 373.112,A -85,B 0,C 180,E1 -27049.991,E2 -27049.991} C_VEL
LIN {X 0,Y 105.66,Z 377.616,A -85,B 0,C 180,E1 -27053.229,E2 -27053.229} C_VEL
LIN {X 0,Y 100.769,Z 383.108,A -85,B 0,C 180,E1 -27058.462,E2 -27058.462} C_VEL
LIN {X 0,Y 96.768,Z 387.437,A -85,B 0,C 180,E1 -27064.167,E2 -27064.167} C_VEL
LIN {X 0,Y 94.589,Z 389.806,A -85,B 0,C 180,E1 -27068.192,E2 -27068.192} C_VEL
LIN {X 0,Y 93.015,Z 391.613,A -85,B 0,C 180,E1 -27072.409,E2 -27072.409} C_VEL
LIN {X 0,Y 91.17,Z 394.076,A -85,B 0,C 180,E1 -27081.131,E2 -27081.131} C_VEL
LIN {X 0,Y 90.87,Z 394.673,A -85,B 0,C 180,E1 -27085.564,E2 -27085.564} C_VEL
LIN {X 0,Y 90.947,Z 394.835,A -85,B 0,C 180,E1 -27090,E2 -27090} C_VEL
LIN {X 0,Y 90.868,Z 394.673,A -85,B 0,C 180,E1 -27094.436,E2 -27094.436} C_VEL
LIN {X 0,Y 91.143,Z 394.075,A -85,B 0,C 180,E1 -27098.871,E2 -27098.871} C_VEL
LIN {X 0,Y 92.991,Z 391.612,A -85,B 0,C 180,E1 -27107.596,E2 -27107.596} C_VEL
LIN {X 0,Y 95.615,Z 388.654,A -85,B 0,C 180,E1 -27113.845,E2 -27113.845} C_VEL
LIN {X 0,Y 99.344,Z 384.663,A -85,B 0,C 180,E1 -27119.683,E2 -27119.683} C_VEL
LIN {X 0,Y 104.033,Z 379.535,A -85,B 0,C 180,E1 -27125.044,E2 -27125.044} C_VEL
LIN {X 0,Y 109.307,Z 373.112,A -85,B 0,C 180,E1 -27130.012,E2 -27130.012} C_VEL
LIN {X 0,Y 114.323,Z 366.574,A -85,B 0,C 180,E1 -27133.755,E2 -27133.755} C_VEL
LIN {X 0,Y 116.224,Z 361.947,A -85,B 0,C 180,E1 -27136.52,E2 -27136.52} C_VEL
LIN {X 0,Y 118.368,Z 354.918,A -85,B 0,C 180,E1 -27140.52,E2 -27140.52} C_VEL
LIN {X 0,Y 119.637,Z 348.687,A -85,B 0,C 180,E1 -27144.003,E2 -27144.003} C_VEL
LIN {X 0,Y 120.019,Z 342.954,A -85,B 0,C 180,E1 -27147.411,E2 -27147.411} C_VEL
LIN {X 0,Y 119.402,Z 338.081,A -85,B 0,C 180,E1 -27150.928,E2 -27150.928} C_VEL
LIN {X 0,Y 118.33,Z 332.856,A -85,B 0,C 180,E1 -27155.413,E2 -27155.413} C_VEL
LIN {X 0,Y 116.965,Z 327.523,A -85,B 0,C 180,E1 -27160.682,E2 -27160.682} C_VEL
LIN {X 0,Y 115.709,Z 323.379,A -85,B 0,C 180,E1 -27166.36,E2 -27166.36} C_VEL
LIN {X 0,Y 115.045,Z 321.903,A -85,B 0,C 180,E1 -27169.42,E2 -27169.42} C_VEL
LIN {X 0,Y 114.244,Z 318.689,A -85,B 0,C 180,E1 -27179.979,E2 -27179.979} C_VEL
LIN {X 0,Y 114.803,Z 321.997,A -85,B 0,C 180,E1 -27191.633,E2 -27191.633} C_VEL
LIN {X 0,Y 115.28,Z 323.04,A -85,B 0,C 180,E1 -27194.092,E2 -27194.092} C_VEL
LIN {X 0,Y 117.178,Z 327.227,A -85,B 0,C 180,E1 -27201.069,E2 -27201.069} C_VEL
LIN {X 0,Y 118.349,Z 330.065,A -85,B 0,C 180,E1 -27204.539,E2 -27204.539} C_VEL
LIN {X 0,Y 119.517,Z 333.322,A -85,B 0,C 180,E1 -27208.112,E2 -27208.112} C_VEL
LIN {X 0,Y 121.152,Z 338.997,A -85,B 0,C 180,E1 -27213.172,E2 -27213.172} C_VEL
LIN {X 0,Y 122.206,Z 343.892,A -85,B 0,C 180,E1 -27217.117,E2 -27217.117} C_VEL
LIN {X 0,Y 123.001,Z 349.367,A -85,B 0,C 180,E1 -27221.217,E2 -27221.217} C_VEL
LIN {X 0,Y 123.345,Z 353.913,A -85,B 0,C 180,E1 -27224.417,E2 -27224.417} C_VEL
LIN {X 0,Y 123.234,Z 360.938,A -85,B 0,C 180,E1 -27229.463,E2 -27229.463} C_VEL
LIN {X 0,Y 122.961,Z 368.051,A -85,B 0,C 180,E1 -27235.142,E2 -27235.142} C_VEL
LIN {X 0,Y 122.991,Z 368.463,A -85,B 0,C 180,E1 -27235.52,E2 -27235.52} C_VEL
LIN {X 0,Y 122.689,Z 371.36,A -85,B 0,C 180,E1 -27237.959,E2 -27237.959} C_VEL
LIN {X 0,Y 121.001,Z 375.892,A -85,B 0,C 180,E1 -27242.034,E2 -27242.034} C_VEL
LIN {X 0,Y 120.113,Z 379.755,A -85,B 0,C 180,E1 -27246.304,E2 -27246.304} C_VEL
LIN {X 0,Y 121.047,Z 381.481,A -85,B 0,C 180,E1 -27248.919,E2 -27248.919} C_VEL
LIN {X 0,Y 124.914,Z 384.112,A -85,B 0,C 180,E1 -27253.662,E2 -27253.662} C_VEL
LIN {X 0,Y 129.4,Z 385.883,A -85,B 0,C 180,E1 -27257.753,E2 -27257.753} C_VEL
LIN {X 0,Y 139.194,Z 387.809,A -85,B 0,C 180,E1 -27264.204,E2 -27264.204} C_VEL
LIN {X 0,Y 147.599,Z 388.299,A -85,B 0,C 180,E1 -27268.345,E2 -27268.345} C_VEL
LIN {X 0,Y 151.501,Z 388.194,A -85,B 0,C 180,E1 -27270,E2 -27270} C_VEL
LIN {X 0,Y 141.006,Z 387.941,A -85,B 0,C 180,E1 -27274.805,E2 -27274.805} C_VEL
LIN {X 0,Y 133.728,Z 386.937,A -85,B 0,C 180,E1 -27279.071,E2 -27279.071} C_VEL
LIN {X 0,Y 128.965,Z 385.731,A -85,B 0,C 180,E1 -27282.59,E2 -27282.59} C_VEL
LIN {X 0,Y 123.166,Z 383.052,A -85,B 0,C 180,E1 -27288.288,E2 -27288.288} C_VEL
LIN {X 0,Y 119.074,Z 379.324,A -85,B 0,C 180,E1 -27294.403,E2 -27294.403} C_VEL
LIN {X 0,Y 116.843,Z 374.655,A -85,B 0,C 180,E1 -27300.521,E2 -27300.521} C_VEL
LIN {X 0,Y 116.254,Z 369.392,A -85,B 0,C 180,E1 -27306.115,E2 -27306.115} C_VEL
LIN {X 0,Y 116.824,Z 363.279,A -85,B 0,C 180,E1 -27311.432,E2 -27311.432} C_VEL
LIN {X 0,Y 117.14,Z 358.87,A -85,B 0,C 180,E1 -27315,E2 -27315} C_VEL
LIN {X 0,Y 117.126,Z 352.456,A -85,B 0,C 180,E1 -27320.085,E2 -27320.085} C_VEL
LIN {X 0,Y 116.534,Z 346.464,A -85,B 0,C 180,E1 -27325.072,E2 -27325.072} C_VEL
LIN {X 0,Y 115.682,Z 342.165,A -85,B 0,C 180,E1 -27328.933,E2 -27328.933} C_VEL
LIN {X 0,Y 114.737,Z 337.997,A -85,B 0,C 180,E1 -27333.235,E2 -27333.235} C_VEL
LIN {X 0,Y 113.319,Z 333.726,A -85,B 0,C 180,E1 -27338.477,E2 -27338.477} C_VEL
LIN {X 0,Y 112.596,Z 331.495,A -85,B 0,C 180,E1 -27341.838,E2 -27341.838} C_VEL
LIN {X 0,Y 111.887,Z 329.529,A -85,B 0,C 180,E1 -27345.471,E2 -27345.471} C_VEL
LIN {X 0,Y 111.244,Z 328.005,A -85,B 0,C 180,E1 -27349.097,E2 -27349.097} C_VEL
LIN {X 0,Y 111.09,Z 325.146,A -85,B 0,C 180,E1 -27360.021,E2 -27360.021} C_VEL
LIN {X 0,Y 111.672,Z 328.383,A -85,B 0,C 180,E1 -27370.904,E2 -27370.904} C_VEL
LIN {X 0,Y 111.941,Z 329.077,A -85,B 0,C 180,E1 -27372.412,E2 -27372.412} C_VEL
LIN {X 0,Y 112.904,Z 332.966,A -85,B 0,C 180,E1 -27378.155,E2 -27378.155} C_VEL
LIN {X 0,Y 113.512,Z 336.09,A -85,B 0,C 180,E1 -27381.828,E2 -27381.828} C_VEL
LIN {X 0,Y 114.325,Z 341.172,A -85,B 0,C 180,E1 -27386.632,E2 -27386.632} C_VEL
LIN {X 0,Y 114.692,Z 346.317,A -85,B 0,C 180,E1 -27390.923,E2 -27390.923} C_VEL
LIN {X 0,Y 114.354,Z 350.363,A -85,B 0,C 180,E1 -27393.604,E2 -27393.604} C_VEL
LIN {X 0,Y 112.9,Z 356.265,A -85,B 0,C 180,E1 -27397.184,E2 -27397.184} C_VEL
LIN {X 0,Y 109.753,Z 364.968,A -85,B 0,C 180,E1 -27402.576,E2 -27402.576} C_VEL
LIN {X 0,Y 108.218,Z 367.756,A -85,B 0,C 180,E1 -27404.41,E2 -27404.41} C_VEL
LIN {X 0,Y 102.826,Z 374.188,A -85,B 0,C 180,E1 -27408.343,E2 -27408.343} C_VEL
LIN {X 0,Y 98.233,Z 379.338,A -85,B 0,C 180,E1 -27412.547,E2 -27412.547} C_VEL
LIN {X 0,Y 93.199,Z 384.467,A -85,B 0,C 180,E1 -27418.14,E2 -27418.14} C_VEL
LIN {X 0,Y 89.141,Z 388.459,A -85,B 0,C 180,E1 -27424.303,E2 -27424.303} C_VEL
LIN {X 0,Y 86.248,Z 391.417,A -85,B 0,C 180,E1 -27430.978,E2 -27430.978} C_VEL
LIN {X 0,Y 84.157,Z 393.881,A -85,B 0,C 180,E1 -27440.386,E2 -27440.386} C_VEL
LIN {X 0,Y 83.796,Z 394.478,A -85,B 0,C 180,E1 -27445.189,E2 -27445.189} C_VEL
LIN {X 0,Y 83.845,Z 394.64,A -85,B 0,C 180,E1 -27450,E2 -27450} C_VEL
LIN {X 0,Y 83.793,Z 394.478,A -85,B 0,C 180,E1 -27454.811,E2 -27454.811} C_VEL
LIN {X 0,Y 84.108,Z 393.88,A -85,B 0,C 180,E1 -27459.62,E2 -27459.62} C_VEL
LIN {X 0,Y 86.228,Z 391.417,A -85,B 0,C 180,E1 -27469.027,E2 -27469.027} C_VEL
LIN {X 0,Y 89.141,Z 388.459,A -85,B 0,C 180,E1 -27475.697,E2 -27475.697} C_VEL
LIN {X 0,Y 93.201,Z 384.467,A -85,B 0,C 180,E1 -27481.859,E2 -27481.859} C_VEL
LIN {X 0,Y 98.273,Z 379.339,A -85,B 0,C 180,E1 -27487.435,E2 -27487.435} C_VEL
LIN {X 0,Y 102.843,Z 374.188,A -85,B 0,C 180,E1 -27491.649,E2 -27491.649} C_VEL
LIN {X 0,Y 108.179,Z 367.755,A -85,B 0,C 180,E1 -27495.611,E2 -27495.611} C_VEL
LIN {X 0,Y 109.749,Z 364.968,A -85,B 0,C 180,E1 -27497.426,E2 -27497.426} C_VEL
LIN {X 0,Y 112.914,Z 356.253,A -85,B 0,C 180,E1 -27502.817,E2 -27502.817} C_VEL
LIN {X 0,Y 114.313,Z 350.416,A -85,B 0,C 180,E1 -27506.383,E2 -27506.383} C_VEL
LIN {X 0,Y 114.688,Z 346.317,A -85,B 0,C 180,E1 -27509.08,E2 -27509.08} C_VEL
LIN {X 0,Y 114.34,Z 341.145,A -85,B 0,C 180,E1 -27513.375,E2 -27513.375} C_VEL
LIN {X 0,Y 113.48,Z 336.018,A -85,B 0,C 180,E1 -27518.272,E2 -27518.272} C_VEL
LIN {X 0,Y 112.939,Z 332.909,A -85,B 0,C 180,E1 -27521.851,E2 -27521.851} C_VEL
LIN {X 0,Y 111.945,Z 329.07,A -85,B 0,C 180,E1 -27527.589,E2 -27527.589} C_VEL
LIN {X 0,Y 111.093,Z 327.191,A -85,B 0,C 180,E1 -27532.71,E2 -27532.71} C_VEL
LIN {X 0,Y 111.085,Z 325.156,A -85,B 0,C 180,E1 -27539.979,E2 -27539.979} C_VEL
LIN {X 0,Y 111.242,Z 328.01,A -85,B 0,C 180,E1 -27550.903,E2 -27550.903} C_VEL
LIN {X 0,Y 111.854,Z 329.591,A -85,B 0,C 180,E1 -27554.533,E2 -27554.533} C_VEL
LIN {X 0,Y 113.045,Z 332.722,A -85,B 0,C 180,E1 -27560.161,E2 -27560.161} C_VEL
LIN {X 0,Y 113.881,Z 335.275,A -85,B 0,C 180,E1 -27563.625,E2 -27563.625} C_VEL
LIN {X 0,Y 115.022,Z 339.26,A -85,B 0,C 180,E1 -27568.102,E2 -27568.102} C_VEL
LIN {X 0,Y 116.134,Z 344.209,A -85,B 0,C 180,E1 -27572.974,E2 -27572.974} C_VEL
LIN {X 0,Y 116.78,Z 348.821,A -85,B 0,C 180,E1 -27576.972,E2 -27576.972} C_VEL
LIN {X 0,Y 117.218,Z 354.114,A -85,B 0,C 180,E1 -27581.234,E2 -27581.234} C_VEL
LIN {X 0,Y 117.104,Z 360.226,A -85,B 0,C 180,E1 -27586.037,E2 -27586.037} C_VEL
LIN {X 0,Y 116.432,Z 367.034,A -85,B 0,C 180,E1 -27591.655,E2 -27591.655} C_VEL
LIN {X 0,Y 116.526,Z 373.004,A -85,B 0,C 180,E1 -27597.562,E2 -27597.562} C_VEL
LIN {X 0,Y 118.044,Z 377.646,A -85,B 0,C 180,E1 -27603.208,E2 -27603.208} C_VEL
LIN {X 0,Y 121.047,Z 381.481,A -85,B 0,C 180,E1 -27608.919,E2 -27608.919} C_VEL
LIN {X 0,Y 122.324,Z 383.088,A -85,B 0,C 180,E1 -27611.549,E2 -27611.549} C_VEL
LIN {X 0,Y 123.988,Z 386.329,A -85,B 0,C 180,E1 -27617.785,E2 -27617.785} C_VEL
LIN {X 0,Y 126.173,Z 387.485,A -85,B 0,C 180,E1 -27621.194,E2 -27621.194} C_VEL
LIN {X 0,Y 128.065,Z 387.859,A -85,B 0,C 180,E1 -27622.726,E2 -27622.726} C_VEL
LIN {X 0,Y 135.494,Z 388.479,A -85,B 0,C 180,E1 -27627.027,E2 -27627.027} C_VEL
LIN {X 0,Y 141.827,Z 388.454,A -85,B 0,C 180,E1 -27630,E2 -27630} C_VEL
LIN {X 0,Y 133.786,Z 388.365,A -85,B 0,C 180,E1 -27633.862,E2 -27633.862} C_VEL
LIN {X 0,Y 127.568,Z 387.803,A -85,B 0,C 180,E1 -27637.574,E2 -27637.574} C_VEL
LIN {X 0,Y 120.038,Z 385.983,A -85,B 0,C 180,E1 -27643.544,E2 -27643.544} C_VEL
LIN {X 0,Y 114.733,Z 383.324,A -85,B 0,C 180,E1 -27649.642,E2 -27649.642} C_VEL
LIN {X 0,Y 112.216,Z 381.008,A -85,B 0,C 180,E1 -27654.021,E2 -27654.021} C_VEL
LIN {X 0,Y 110.014,Z 376.512,A -85,B 0,C 180,E1 -27660.734,E2 -27660.734} C_VEL
LIN {X 0,Y 109.658,Z 370.731,A -85,B 0,C 180,E1 -27667.506,E2 -27667.506} C_VEL
LIN {X 0,Y 110.547,Z 364.839,A -85,B 0,C 180,E1 -27673.11,E2 -27673.11} C_VEL
LIN {X 0,Y 111.101,Z 358.884,A -85,B 0,C 180,E1 -27678.403,E2 -27678.403} C_VEL
LIN {X 0,Y 111.186,Z 353.637,A -85,B 0,C 180,E1 -27683.124,E2 -27683.124} C_VEL
LIN {X 0,Y 110.769,Z 348.566,A -85,B 0,C 180,E1 -27687.883,E2 -27687.883} C_VEL
LIN {X 0,Y 109.94,Z 343.356,A -85,B 0,C 180,E1 -27693.5,E2 -27693.5} C_VEL
LIN {X 0,Y 109.043,Z 339.435,A -85,B 0,C 180,E1 -27698.762,E2 -27698.762} C_VEL
LIN {X 0,Y 108.298,Z 336.804,A -85,B 0,C 180,E1 -27703.044,E2 -27703.044} C_VEL
LIN {X 0,Y 107.514,Z 334.262,A -85,B 0,C 180,E1 -27708.714,E2 -27708.714} C_VEL
LIN {X 0,Y 107.642,Z 331.442,A -85,B 0,C 180,E1 -27720.022,E2 -27720.022} C_VEL
LIN {X 0,Y 108.009,Z 334.669,A -85,B 0,C 180,E1 -27731.278,E2 -27731.278} C_VEL
LIN {X 0,Y 108.572,Z 338.136,A -85,B 0,C 180,E1 -27736.957,E2 -27736.957} C_VEL
LIN {X 0,Y 109.111,Z 342.989,A -85,B 0,C 180,E1 -27742.757,E2 -27742.757} C_VEL
LIN {X 0,Y 109.421,Z 348.129,A -85,B 0,C 180,E1 -27747.775,E2 -27747.775} C_VEL
LIN {X 0,Y 109.111,Z 352.083,A -85,B 0,C 180,E1 -27751.04,E2 -27751.04} C_VEL
LIN {X 0,Y 107.364,Z 358.196,A -85,B 0,C 180,E1 -27755.084,E2 -27755.084} C_VEL
LIN {X 0,Y 103.922,Z 366.159,A -85,B 0,C 180,E1 -27760.466,E2 -27760.466} C_VEL
LIN {X 0,Y 103.206,Z 367.555,A -85,B 0,C 180,E1 -27761.492,E2 -27761.492} C_VEL
LIN {X 0,Y 98.814,Z 372.721,A -85,B 0,C 180,E1 -27764.666,E2 -27764.666} C_VEL
LIN {X 0,Y 94.593,Z 377.223,A -85,B 0,C 180,E1 -27768.036,E2 -27768.036} C_VEL
LIN {X 0,Y 88.94,Z 382.718,A -85,B 0,C 180,E1 -27773.656,E2 -27773.656} C_VEL
LIN {X 0,Y 84.152,Z 387.045,A -85,B 0,C 180,E1 -27779.928,E2 -27779.928} C_VEL
LIN {X 0,Y 81.51,Z 389.415,A -85,B 0,C 180,E1 -27784.463,E2 -27784.463} C_VEL
LIN {X 0,Y 79.531,Z 391.222,A -85,B 0,C 180,E1 -27789.301,E2 -27789.301} C_VEL
LIN {X 0,Y 77.146,Z 393.686,A -85,B 0,C 180,E1 -27799.502,E2 -27799.502} C_VEL
LIN {X 0,Y 76.706,Z 394.283,A -85,B 0,C 180,E1 -27804.743,E2 -27804.743} C_VEL
LIN {X 0,Y 76.766,Z 394.446,A -85,B 0,C 180,E1 -27810,E2 -27810} C_VEL
LIN {X 0,Y 76.699,Z 394.283,A -85,B 0,C 180,E1 -27815.257,E2 -27815.257} C_VEL
LIN {X 0,Y 77.102,Z 393.684,A -85,B 0,C 180,E1 -27820.504,E2 -27820.504} C_VEL
LIN {X 0,Y 79.515,Z 391.221,A -85,B 0,C 180,E1 -27830.704,E2 -27830.704} C_VEL
LIN {X 0,Y 82.778,Z 388.264,A -85,B 0,C 180,E1 -27837.837,E2 -27837.837} C_VEL
LIN {X 0,Y 87.216,Z 384.272,A -85,B 0,C 180,E1 -27844.337,E2 -27844.337} C_VEL
LIN {X 0,Y 92.703,Z 379.143,A -85,B 0,C 180,E1 -27850.12,E2 -27850.12} C_VEL
LIN {X 0,Y 97.613,Z 373.992,A -85,B 0,C 180,E1 -27854.441,E2 -27854.441} C_VEL
LIN {X 0,Y 102.163,Z 368.935,A -85,B 0,C 180,E1 -27857.689,E2 -27857.689} C_VEL
LIN {X 0,Y 103.176,Z 367.553,A -85,B 0,C 180,E1 -27858.526,E2 -27858.526} C_VEL
LIN {X 0,Y 106.002,Z 361.515,A -85,B 0,C 180,E1 -27862.711,E2 -27862.711} C_VEL
LIN {X 0,Y 107.94,Z 356.405,A -85,B 0,C 180,E1 -27866.123,E2 -27866.123} C_VEL
LIN {X 0,Y 109.056,Z 352.153,A -85,B 0,C 180,E1 -27868.943,E2 -27868.943} C_VEL
LIN {X 0,Y 109.418,Z 348.134,A -85,B 0,C 180,E1 -27872.224,E2 -27872.224} C_VEL
LIN {X 0,Y 109.259,Z 344.871,A -85,B 0,C 180,E1 -27875.261,E2 -27875.261} C_VEL
LIN {X 0,Y 108.921,Z 340.734,A -85,B 0,C 180,E1 -27879.829,E2 -27879.829} C_VEL
LIN {X 0,Y 108.602,Z 338.088,A -85,B 0,C 180,E1 -27883.048,E2 -27883.048} C_VEL
LIN {X 0,Y 108.009,Z 334.669,A -85,B 0,C 180,E1 -27888.722,E2 -27888.722} C_VEL
LIN {X 0,Y 107.629,Z 331.462,A -85,B 0,C 180,E1 -27899.978,E2 -27899.978} C_VEL
LIN {X 0,Y 107.202,Z 333.158,A -85,B 0,C 180,E1 -27907.523,E2 -27907.523} C_VEL
LIN {X 0,Y 107.512,Z 334.287,A -85,B 0,C 180,E1 -27911.33,E2 -27911.33} C_VEL
LIN {X 0,Y 107.964,Z 335.886,A -85,B 0,C 180,E1 -27915.069,E2 -27915.069} C_VEL
LIN {X 0,Y 108.659,Z 337.867,A -85,B 0,C 180,E1 -27918.844,E2 -27918.844} C_VEL
LIN {X 0,Y 109.295,Z 340.376,A -85,B 0,C 180,E1 -27922.67,E2 -27922.67} C_VEL
LIN {X 0,Y 109.944,Z 343.41,A -85,B 0,C 180,E1 -27926.555,E2 -27926.555} C_VEL
LIN {X 0,Y 110.796,Z 348.54,A -85,B 0,C 180,E1 -27932.115,E2 -27932.115} C_VEL
LIN {X 0,Y 111.204,Z 353.614,A -85,B 0,C 180,E1 -27936.869,E2 -27936.869} C_VEL
LIN {X 0,Y 111.157,Z 358.825,A -85,B 0,C 180,E1 -27941.58,E2 -27941.58} C_VEL
LIN {X 0,Y 110.539,Z 364.839,A -85,B 0,C 180,E1 -27946.886,E2 -27946.886} C_VEL
LIN {X 0,Y 109.61,Z 371.845,A -85,B 0,C 180,E1 -27953.624,E2 -27953.624} C_VEL
LIN {X 0,Y 110.507,Z 377.843,A -85,B 0,C 180,E1 -27961.166,E2 -27961.166} C_VEL
LIN {X 0,Y 112.227,Z 381.007,A -85,B 0,C 180,E1 -27965.981,E2 -27965.981} C_VEL
LIN {X 0,Y 117.231,Z 384.783,A -85,B 0,C 180,E1 -27973.494,E2 -27973.494} C_VEL
LIN {X 0,Y 121.992,Z 386.648,A -85,B 0,C 180,E1 -27978.231,E2 -27978.231} C_VEL
LIN {X 0,Y 128.065,Z 387.859,A -85,B 0,C 180,E1 -27982.726,E2 -27982.726} C_VEL
LIN {X 0,Y 129.936,Z 388.211,A -85,B 0,C 180,E1 -27984.424,E2 -27984.424} C_VEL
LIN {X 0,Y 130.855,Z 388.549,A -85,B 0,C 180,E1 -27986.267,E2 -27986.267} C_VEL
LIN {X 0,Y 130.979,Z 388.752,A -85,B 0,C 180,E1 -27988.146,E2 -27988.146} C_VEL
LIN {X 0,Y 130.082,Z 388.785,A -85,B 0,C 180,E1 -27990.283,E2 -27990.283} C_VEL
LIN {X 0,Y 128.221,Z 388.827,A -85,B 0,C 180,E1 -27991.945,E2 -27991.945} C_VEL
LIN {X 0,Y 127.79,Z 388.772,A -85,B 0,C 180,E1 -27992.192,E2 -27992.192} C_VEL
LIN {X 0,Y 120.262,Z 388.324,A -85,B 0,C 180,E1 -27996.754,E2 -27996.754} C_VEL
LIN {X 0,Y 114.594,Z 387.27,A -85,B 0,C 180,E1 -28001.229,E2 -28001.229} C_VEL
LIN {X 0,Y 107.815,Z 384.604,A -85,B 0,C 180,E1 -28009.021,E2 -28009.021} C_VEL
LIN {X 0,Y 104.442,Z 381.266,A -85,B 0,C 180,E1 -28015.9,E2 -28015.9} C_VEL
LIN {X 0,Y 102.88,Z 376.742,A -85,B 0,C 180,E1 -28023.126,E2 -28023.126} C_VEL
LIN {X 0,Y 103.221,Z 371.354,A -85,B 0,C 180,E1 -28029.847,E2 -28029.847} C_VEL
LIN {X 0,Y 104.334,Z 366.398,A -85,B 0,C 180,E1 -28035.013,E2 -28035.013} C_VEL
LIN {X 0,Y 105.118,Z 360.763,A -85,B 0,C 180,E1 -28040.6,E2 -28040.6} C_VEL
LIN {X 0,Y 105.349,Z 356.314,A -85,B 0,C 180,E1 -28044.97,E2 -28044.97} C_VEL
LIN {X 0,Y 105.292,Z 352.529,A -85,B 0,C 180,E1 -28049.047,E2 -28049.047} C_VEL
LIN {X 0,Y 104.852,Z 347.736,A -85,B 0,C 180,E1 -28054.889,E2 -28054.889} C_VEL
LIN {X 0,Y 104.238,Z 344.046,A -85,B 0,C 180,E1 -28060.324,E2 -28060.324} C_VEL
LIN {X 0,Y 103.8,Z 341.944,A -85,B 0,C 180,E1 -28064.311,E2 -28064.311} C_VEL
LIN {X 0,Y 103.486,Z 340.345,A -85,B 0,C 180,E1 -28068.268,E2 -28068.268} C_VEL
LIN {X 0,Y 103.31,Z 338.272,A -85,B 0,C 180,E1 -28076.122,E2 -28076.122} C_VEL
LIN {X 0,Y 103.718,Z 337.475,A -85,B 0,C 180,E1 -28080.023,E2 -28080.023} C_VEL
LIN {X 0,Y 103.612,Z 339.499,A -85,B 0,C 180,E1 -28087.819,E2 -28087.819} C_VEL
LIN {X 0,Y 103.93,Z 340.937,A -85,B 0,C 180,E1 -28091.727,E2 -28091.727} C_VEL
LIN {X 0,Y 104.054,Z 343.175,A -85,B 0,C 180,E1 -28095.697,E2 -28095.697} C_VEL
LIN {X 0,Y 104.178,Z 346.092,A -85,B 0,C 180,E1 -28099.736,E2 -28099.736} C_VEL
LIN {X 0,Y 104.249,Z 349.697,A -85,B 0,C 180,E1 -28103.882,E2 -28103.882} C_VEL
LIN {X 0,Y 103.867,Z 354.209,A -85,B 0,C 180,E1 -28108.406,E2 -28108.406} C_VEL
LIN {X 0,Y 103.445,Z 356.102,A -85,B 0,C 180,E1 -28109.898,E2 -28109.898} C_VEL
LIN {X 0,Y 101.305,Z 361.378,A -85,B 0,C 180,E1 -28113.736,E2 -28113.736} C_VEL
LIN {X 0,Y 98.238,Z 367.342,A -85,B 0,C 180,E1 -28118.101,E2 -28118.101} C_VEL
LIN {X 0,Y 97.469,Z 368.738,A -85,B 0,C 180,E1 -28119.185,E2 -28119.185} C_VEL
LIN {X 0,Y 90.512,Z 375.991,A -85,B 0,C 180,E1 -28124.092,E2 -28124.092} C_VEL
LIN {X 0,Y 83.314,Z 382.523,A -85,B 0,C 180,E1 -28130.754,E2 -28130.754} C_VEL
LIN {X 0,Y 78.067,Z 386.85,A -85,B 0,C 180,E1 -28137.307,E2 -28137.307} C_VEL
LIN {X 0,Y 75.14,Z 389.219,A -85,B 0,C 180,E1 -28142.118,E2 -28142.118} C_VEL
LIN {X 0,Y 72.903,Z 391.026,A -85,B 0,C 180,E1 -28147.319,E2 -28147.319} C_VEL
LIN {X 0,Y 70.145,Z 393.49,A -85,B 0,C 180,E1 -28158.441,E2 -28158.441} C_VEL
LIN {X 0,Y 69.625,Z 394.088,A -85,B 0,C 180,E1 -28164.207,E2 -28164.207} C_VEL
LIN {X 0,Y 69.676,Z 394.252,A -85,B 0,C 180,E1 -28170,E2 -28170} C_VEL
LIN {X 0,Y 69.616,Z 394.088,A -85,B 0,C 180,E1 -28175.794,E2 -28175.794} C_VEL
LIN {X 0,Y 70.106,Z 393.489,A -85,B 0,C 180,E1 -28181.566,E2 -28181.566} C_VEL
LIN {X 0,Y 72.872,Z 391.025,A -85,B 0,C 180,E1 -28192.691,E2 -28192.691} C_VEL
LIN {X 0,Y 76.552,Z 388.068,A -85,B 0,C 180,E1 -28200.326,E2 -28200.326} C_VEL
LIN {X 0,Y 81.424,Z 384.076,A -85,B 0,C 180,E1 -28207.17,E2 -28207.17} C_VEL
LIN {X 0,Y 86.775,Z 379.498,A -85,B 0,C 180,E1 -28212.592,E2 -28212.592} C_VEL
LIN {X 0,Y 92.767,Z 373.681,A -85,B 0,C 180,E1 -28217.616,E2 -28217.616} C_VEL
LIN {X 0,Y 97.424,Z 368.736,A -85,B 0,C 180,E1 -28220.847,E2 -28220.847} C_VEL
LIN {X 0,Y 100.713,Z 362.647,A -85,B 0,C 180,E1 -28225.397,E2 -28225.397} C_VEL
LIN {X 0,Y 102.757,Z 357.974,A -85,B 0,C 180,E1 -28228.75,E2 -28228.75} C_VEL
LIN {X 0,Y 103.866,Z 354.102,A -85,B 0,C 180,E1 -28231.705,E2 -28231.705} C_VEL
LIN {X 0,Y 104.24,Z 349.708,A -85,B 0,C 180,E1 -28236.115,E2 -28236.115} C_VEL
LIN {X 0,Y 104.101,Z 344.568,A -85,B 0,C 180,E1 -28242.289,E2 -28242.289} C_VEL
LIN {X 0,Y 104.103,Z 343.11,A -85,B 0,C 180,E1 -28244.311,E2 -28244.311} C_VEL
LIN {X 0,Y 103.96,Z 340.897,A -85,B 0,C 180,E1 -28248.276,E2 -28248.276} C_VEL
LIN {X 0,Y 103.609,Z 339.503,A -85,B 0,C 180,E1 -28252.181,E2 -28252.181} C_VEL
LIN {X 0,Y 103.713,Z 337.484,A -85,B 0,C 180,E1 -28259.977,E2 -28259.977} C_VEL
LIN {X 0,Y 103.287,Z 339.191,A -85,B 0,C 180,E1 -28267.798,E2 -28267.798} C_VEL
LIN {X 0,Y 103.46,Z 340.379,A -85,B 0,C 180,E1 -28271.735,E2 -28271.735} C_VEL
LIN {X 0,Y 103.756,Z 342.003,A -85,B 0,C 180,E1 -28275.696,E2 -28275.696} C_VEL
LIN {X 0,Y 104.492,Z 345.308,A -85,B 0,C 180,E1 -28281.685,E2 -28281.685} C_VEL
LIN {X 0,Y 105.033,Z 349.916,A -85,B 0,C 180,E1 -28287.902,E2 -28287.902} C_VEL
LIN {X 0,Y 105.404,Z 353.676,A -85,B 0,C 180,E1 -28292.208,E2 -28292.208} C_VEL
LIN {X 0,Y 105.236,Z 359.396,A -85,B 0,C 180,E1 -28298.12,E2 -28298.12} C_VEL
LIN {X 0,Y 104.639,Z 364.46,A -85,B 0,C 180,E1 -28303.139,E2 -28303.139} C_VEL
LIN {X 0,Y 103.579,Z 369.544,A -85,B 0,C 180,E1 -28308.239,E2 -28308.239} C_VEL
LIN {X 0,Y 102.853,Z 374.457,A -85,B 0,C 180,E1 -28313.906,E2 -28313.906} C_VEL
LIN {X 0,Y 103.182,Z 378.322,A -85,B 0,C 180,E1 -28319.281,E2 -28319.281} C_VEL
LIN {X 0,Y 105.313,Z 382.403,A -85,B 0,C 180,E1 -28326.397,E2 -28326.397} C_VEL
LIN {X 0,Y 107.853,Z 384.603,A -85,B 0,C 180,E1 -28330.986,E2 -28330.986} C_VEL
LIN {X 0,Y 114.595,Z 387.268,A -85,B 0,C 180,E1 -28338.767,E2 -28338.767} C_VEL
LIN {X 0,Y 122.314,Z 388.476,A -85,B 0,C 180,E1 -28344.587,E2 -28344.587} C_VEL
LIN {X 0,Y 132.136,Z 388.719,A -85,B 0,C 180,E1 -28350,E2 -28350} C_VEL
LIN {X 0,Y 127.79,Z 388.772,A -85,B 0,C 180,E1 -28352.192,E2 -28352.192} C_VEL
LIN {X 0,Y 123.59,Z 388.785,A -85,B 0,C 180,E1 -28354.089,E2 -28354.089} C_VEL
LIN {X 0,Y 109.68,Z 388.12,A -85,B 0,C 180,E1 -28359.567,E2 -28359.567} C_VEL
LIN {X 0,Y 105.496,Z 387.46,A -85,B 0,C 180,E1 -28362.434,E2 -28362.434} C_VEL
LIN {X 0,Y 105.043,Z 387.286,A -85,B 0,C 180,E1 -28362.902,E2 -28362.902} C_VEL
LIN {X 0,Y 99.58,Z 384.844,A -85,B 0,C 180,E1 -28370.663,E2 -28370.663} C_VEL
LIN {X 0,Y 96.55,Z 380.912,A -85,B 0,C 180,E1 -28379.189,E2 -28379.189} C_VEL
LIN {X 0,Y 96.057,Z 376.524,A -85,B 0,C 180,E1 -28386.454,E2 -28386.454} C_VEL
LIN {X 0,Y 97.336,Z 370.782,A -85,B 0,C 180,E1 -28393.816,E2 -28393.816} C_VEL
LIN {X 0,Y 98.397,Z 366.987,A -85,B 0,C 180,E1 -28398.161,E2 -28398.161} C_VEL
LIN {X 0,Y 99.357,Z 361.533,A -85,B 0,C 180,E1 -28404.194,E2 -28404.194} C_VEL
LIN {X 0,Y 99.679,Z 357.19,A -85,B 0,C 180,E1 -28409.172,E2 -28409.172} C_VEL
LIN {X 0,Y 99.666,Z 352.827,A -85,B 0,C 180,E1 -28414.998,E2 -28414.998} C_VEL
LIN {X 0,Y 99.401,Z 349.035,A -85,B 0,C 180,E1 -28421.134,E2 -28421.134} C_VEL
LIN {X 0,Y 99.048,Z 346.188,A -85,B 0,C 180,E1 -28427.735,E2 -28427.735} C_VEL
LIN {X 0,Y 99.005,Z 344.036,A -85,B 0,C 180,E1 -28435.953,E2 -28435.953} C_VEL
LIN {X 0,Y 99.493,Z 343.281,A -85,B 0,C 180,E1 -28440.024,E2 -28440.024} C_VEL
LIN {X 0,Y 99.238,Z 345.291,A -85,B 0,C 180,E1 -28448.166,E2 -28448.166} C_VEL
LIN {X 0,Y 99.397,Z 346.907,A -85,B 0,C 180,E1 -28452.27,E2 -28452.27} C_VEL
LIN {X 0,Y 99.317,Z 349.4,A -85,B 0,C 180,E1 -28456.466,E2 -28456.466} C_VEL
LIN {X 0,Y 99.115,Z 352.403,A -85,B 0,C 180,E1 -28460.789,E2 -28460.789} C_VEL
LIN {X 0,Y 98.712,Z 356.322,A -85,B 0,C 180,E1 -28465.314,E2 -28465.314} C_VEL
LIN {X 0,Y 98.188,Z 358.299,A -85,B 0,C 180,E1 -28467.302,E2 -28467.302} C_VEL
LIN {X 0,Y 96.23,Z 362.628,A -85,B 0,C 180,E1 -28470.772,E2 -28470.772} C_VEL
LIN {X 0,Y 92.755,Z 368.525,A -85,B 0,C 180,E1 -28475.462,E2 -28475.462} C_VEL
LIN {X 0,Y 91.877,Z 369.92,A -85,B 0,C 180,E1 -28476.567,E2 -28476.567} C_VEL
LIN {X 0,Y 84.522,Z 376.832,A -85,B 0,C 180,E1 -28481.554,E2 -28481.554} C_VEL
LIN {X 0,Y 77.934,Z 382.328,A -85,B 0,C 180,E1 -28487.443,E2 -28487.443} C_VEL
LIN {X 0,Y 72.176,Z 386.655,A -85,B 0,C 180,E1 -28494.252,E2 -28494.252} C_VEL
LIN {X 0,Y 68.925,Z 389.024,A -85,B 0,C 180,E1 -28499.349,E2 -28499.349} C_VEL
LIN {X 0,Y 64.472,Z 392.227,A -85,B 0,C 180,E1 -28510.912,E2 -28510.912} C_VEL
LIN {X 0,Y 63.187,Z 393.295,A -85,B 0,C 180,E1 -28517.147,E2 -28517.147} C_VEL
LIN {X 0,Y 62.565,Z 393.894,A -85,B 0,C 180,E1 -28523.55,E2 -28523.55} C_VEL
LIN {X 0,Y 62.576,Z 394.057,A -85,B 0,C 180,E1 -28530,E2 -28530} C_VEL
LIN {X 0,Y 62.556,Z 393.893,A -85,B 0,C 180,E1 -28536.45,E2 -28536.45} C_VEL
LIN {X 0,Y 63.152,Z 393.294,A -85,B 0,C 180,E1 -28542.86,E2 -28542.86} C_VEL
LIN {X 0,Y 66.336,Z 390.829,A -85,B 0,C 180,E1 -28555.073,E2 -28555.073} C_VEL
LIN {X 0,Y 70.5,Z 387.873,A -85,B 0,C 180,E1 -28563.248,E2 -28563.248} C_VEL
LIN {X 0,Y 75.867,Z 383.881,A -85,B 0,C 180,E1 -28570.424,E2 -28570.424} C_VEL
LIN {X 0,Y 81.359,Z 379.564,A -85,B 0,C 180,E1 -28575.719,E2 -28575.719} C_VEL
LIN {X 0,Y 86.898,Z 374.641,A -85,B 0,C 180,E1 -28580.202,E2 -28580.202} C_VEL
LIN {X 0,Y 91.84,Z 369.919,A -85,B 0,C 180,E1 -28583.465,E2 -28583.465} C_VEL
LIN {X 0,Y 95.589,Z 363.928,A -85,B 0,C 180,E1 -28588.244,E2 -28588.244} C_VEL
LIN {X 0,Y 97.455,Z 360.013,A -85,B 0,C 180,E1 -28591.256,E2 -28591.256} C_VEL
LIN {X 0,Y 98.148,Z 358.335,A -85,B 0,C 180,E1 -28592.693,E2 -28592.693} C_VEL
LIN {X 0,Y 98.854,Z 355.071,A -85,B 0,C 180,E1 -28596.042,E2 -28596.042} C_VEL
LIN {X 0,Y 99.213,Z 351,A -85,B 0,C 180,E1 -28601.117,E2 -28601.117} C_VEL
LIN {X 0,Y 99.453,Z 347.998,A -85,B 0,C 180,E1 -28605.657,E2 -28605.657} C_VEL
LIN {X 0,Y 99.396,Z 346.908,A -85,B 0,C 180,E1 -28607.73,E2 -28607.73} C_VEL
LIN {X 0,Y 99.228,Z 345.054,A -85,B 0,C 180,E1 -28612.547,E2 -28612.547} C_VEL
LIN {X 0,Y 99.486,Z 343.29,A -85,B 0,C 180,E1 -28619.976,E2 -28619.976} C_VEL
LIN {X 0,Y 98.902,Z 344.942,A -85,B 0,C 180,E1 -28628.146,E2 -28628.146} C_VEL
LIN {X 0,Y 99.01,Z 346.238,A -85,B 0,C 180,E1 -28632.27,E2 -28632.27} C_VEL
LIN {X 0,Y 99.377,Z 349.057,A -85,B 0,C 180,E1 -28638.862,E2 -28638.862} C_VEL
LIN {X 0,Y 99.513,Z 351.774,A -85,B 0,C 180,E1 -28643.352,E2 -28643.352} C_VEL
LIN {X 0,Y 99.716,Z 354.496,A -85,B 0,C 180,E1 -28647.238,E2 -28647.238} C_VEL
LIN {X 0,Y 99.641,Z 358.299,A -85,B 0,C 180,E1 -28652.18,E2 -28652.18} C_VEL
LIN {X 0,Y 99.149,Z 362.821,A -85,B 0,C 180,E1 -28657.309,E2 -28657.309} C_VEL
LIN {X 0,Y 98.407,Z 366.981,A -85,B 0,C 180,E1 -28661.838,E2 -28661.838} C_VEL
LIN {X 0,Y 96.661,Z 373.291,A -85,B 0,C 180,E1 -28669.129,E2 -28669.129} C_VEL
LIN {X 0,Y 96.054,Z 378.552,A -85,B 0,C 180,E1 -28676.719,E2 -28676.719} C_VEL
LIN {X 0,Y 97.499,Z 382.639,A -85,B 0,C 180,E1 -28684.375,E2 -28684.375} C_VEL
LIN {X 0,Y 99.585,Z 384.844,A -85,B 0,C 180,E1 -28689.338,E2 -28689.338} C_VEL
LIN {X 0,Y 102.577,Z 386.477,A -85,B 0,C 180,E1 -28694.095,E2 -28694.095} C_VEL
LIN {X 0,Y 111.109,Z 388.584,A -85,B 0,C 180,E1 -28702.732,E2 -28702.732} C_VEL
LIN {X 0,Y 119.48,Z 389.067,A -85,B 0,C 180,E1 -28708.295,E2 -28708.295} C_VEL
LIN {X 0,Y 122.582,Z 388.981,A -85,B 0,C 180,E1 -28710,E2 -28710} C_VEL
LIN {X 0,Y 112.983,Z 388.74,A -85,B 0,C 180,E1 -28715.823,E2 -28715.823} C_VEL
LIN {X 0,Y 105.043,Z 387.286,A -85,B 0,C 180,E1 -28722.902,E2 -28722.902} C_VEL
LIN {X 0,Y 102.031,Z 386.627,A -85,B 0,C 180,E1 -28725.69,E2 -28725.69} C_VEL
LIN {X 0,Y 91.987,Z 384.24,A -85,B 0,C 180,E1 -28734.286,E2 -28734.286} C_VEL
LIN {X 0,Y 90.003,Z 382.991,A -85,B 0,C 180,E1 -28737.679,E2 -28737.679} C_VEL
LIN {X 0,Y 89.686,Z 382.503,A -85,B 0,C 180,E1 -28738.872,E2 -28738.872} C_VEL
LIN {X 0,Y 89.418,Z 377.639,A -85,B 0,C 180,E1 -28748.237,E2 -28748.237} C_VEL
LIN {X 0,Y 91.196,Z 372.054,A -85,B 0,C 180,E1 -28756.125,E2 -28756.125} C_VEL
LIN {X 0,Y 92.59,Z 367.804,A -85,B 0,C 180,E1 -28761.5,E2 -28761.5} C_VEL
LIN {X 0,Y 93.366,Z 364.245,A -85,B 0,C 180,E1 -28765.892,E2 -28765.892} C_VEL
LIN {X 0,Y 94,Z 360.492,A -85,B 0,C 180,E1 -28770.954,E2 -28770.954} C_VEL
LIN {X 0,Y 94.252,Z 356.724,A -85,B 0,C 180,E1 -28776.609,E2 -28776.609} C_VEL
LIN {X 0,Y 94.385,Z 354.598,A -85,B 0,C 180,E1 -28780.451,E2 -28780.451} C_VEL
LIN {X 0,Y 94.224,Z 351.753,A -85,B 0,C 180,E1 -28787.096,E2 -28787.096} C_VEL
LIN {X 0,Y 94.214,Z 350.506,A -85,B 0,C 180,E1 -28791.446,E2 -28791.446} C_VEL
LIN {X 0,Y 95.012,Z 348.881,A -85,B 0,C 180,E1 -28800.025,E2 -28800.025} C_VEL
LIN {X 0,Y 94.564,Z 350.905,A -85,B 0,C 180,E1 -28808.573,E2 -28808.573} C_VEL
LIN {X 0,Y 94.478,Z 352.645,A -85,B 0,C 180,E1 -28812.92,E2 -28812.92} C_VEL
LIN {X 0,Y 94.137,Z 355.295,A -85,B 0,C 180,E1 -28817.4,E2 -28817.4} C_VEL
LIN {X 0,Y 93.499,Z 358.602,A -85,B 0,C 180,E1 -28822.101,E2 -28822.101} C_VEL
LIN {X 0,Y 92.848,Z 360.819,A -85,B 0,C 180,E1 -28824.729,E2 -28824.729} C_VEL
LIN {X 0,Y 91.375,Z 363.905,A -85,B 0,C 180,E1 -28827.51,E2 -28827.51} C_VEL
LIN {X 0,Y 87.48,Z 369.708,A -85,B 0,C 180,E1 -28832.485,E2 -28832.485} C_VEL
LIN {X 0,Y 86.477,Z 370.979,A -85,B 0,C 180,E1 -28833.592,E2 -28833.592} C_VEL
LIN {X 0,Y 79.961,Z 376.636,A -85,B 0,C 180,E1 -28837.72,E2 -28837.72} C_VEL
LIN {X 0,Y 72.85,Z 382.132,A -85,B 0,C 180,E1 -28843.654,E2 -28843.654} C_VEL
LIN {X 0,Y 66.53,Z 386.46,A -85,B 0,C 180,E1 -28850.669,E2 -28850.669} C_VEL
LIN {X 0,Y 62.908,Z 388.829,A -85,B 0,C 180,E1 -28856.043,E2 -28856.043} C_VEL
LIN {X 0,Y 57.766,Z 392.032,A -85,B 0,C 180,E1 -28868.594,E2 -28868.594} C_VEL
LIN {X 0,Y 56.279,Z 393.1,A -85,B 0,C 180,E1 -28875.537,E2 -28875.537} C_VEL
LIN {X 0,Y 55.506,Z 393.699,A -85,B 0,C 180,E1 -28882.726,E2 -28882.726} C_VEL
LIN {X 0,Y 55.493,Z 393.863,A -85,B 0,C 180,E1 -28890,E2 -28890} C_VEL
LIN {X 0,Y 55.496,Z 393.698,A -85,B 0,C 180,E1 -28897.275,E2 -28897.275} C_VEL
LIN {X 0,Y 56.22,Z 393.098,A -85,B 0,C 180,E1 -28904.478,E2 -28904.478} C_VEL
LIN {X 0,Y 59.942,Z 390.633,A -85,B 0,C 180,E1 -28917.968,E2 -28917.968} C_VEL
LIN {X 0,Y 64.669,Z 387.678,A -85,B 0,C 180,E1 -28926.706,E2 -28926.706} C_VEL
LIN {X 0,Y 70.598,Z 383.685,A -85,B 0,C 180,E1 -28934.173,E2 -28934.173} C_VEL
LIN {X 0,Y 77.235,Z 378.785,A -85,B 0,C 180,E1 -28940.171,E2 -28940.171} C_VEL
LIN {X 0,Y 83.803,Z 373.289,A -85,B 0,C 180,E1 -28944.85,E2 -28944.85} C_VEL
LIN {X 0,Y 86.443,Z 370.977,A -85,B 0,C 180,E1 -28946.442,E2 -28946.442} C_VEL
LIN {X 0,Y 89.385,Z 366.91,A -85,B 0,C 180,E1 -28949.868,E2 -28949.868} C_VEL
LIN {X 0,Y 92.274,Z 362.179,A -85,B 0,C 180,E1 -28953.964,E2 -28953.964} C_VEL
LIN {X 0,Y 93.177,Z 359.837,A -85,B 0,C 180,E1 -28956.354,E2 -28956.354} C_VEL
LIN {X 0,Y 93.853,Z 356.914,A -85,B 0,C 180,E1 -28960.282,E2 -28960.282} C_VEL
LIN {X 0,Y 94.374,Z 353.503,A -85,B 0,C 180,E1 -28965.484,E2 -28965.484} C_VEL
LIN {X 0,Y 94.52,Z 352.598,A -85,B 0,C 180,E1 -28967.086,E2 -28967.086} C_VEL
LIN {X 0,Y 94.565,Z 350.904,A -85,B 0,C 180,E1 -28971.427,E2 -28971.427} C_VEL
LIN {X 0,Y 95.007,Z 348.887,A -85,B 0,C 180,E1 -28979.975,E2 -28979.975} C_VEL
LIN {X 0,Y 94.215,Z 350.505,A -85,B 0,C 180,E1 -28988.554,E2 -28988.554} C_VEL
LIN {X 0,Y 94.168,Z 352.229,A -85,B 0,C 180,E1 -28994.024,E2 -28994.024} C_VEL
LIN {X 0,Y 94.379,Z 354.604,A -85,B 0,C 180,E1 -28999.551,E2 -28999.551} C_VEL
LIN {X 0,Y 94.11,Z 358.764,A -85,B 0,C 180,E1 -29006.59,E2 -29006.59} C_VEL
LIN {X 0,Y 93.749,Z 362.364,A -85,B 0,C 180,E1 -29011.62,E2 -29011.62} C_VEL
LIN {X 0,Y 92.868,Z 366.758,A -85,B 0,C 180,E1 -29017.224,E2 -29017.224} C_VEL
LIN {X 0,Y 91.548,Z 370.986,A -85,B 0,C 180,E1 -29022.566,E2 -29022.566} C_VEL
LIN {X 0,Y 89.501,Z 377.195,A -85,B 0,C 180,E1 -29031.084,E2 -29031.084} C_VEL
LIN {X 0,Y 89.479,Z 381.906,A -85,B 0,C 180,E1 -29039.708,E2 -29039.708} C_VEL
LIN {X 0,Y 91.485,Z 385.082,A -85,B 0,C 180,E1 -29047.412,E2 -29047.412} C_VEL
LIN {X 0,Y 94.989,Z 387.166,A -85,B 0,C 180,E1 -29054.017,E2 -29054.017} C_VEL
LIN {X 0,Y 102.006,Z 388.836,A -85,B 0,C 180,E1 -29062.08,E2 -29062.08} C_VEL
LIN {X 0,Y 107.138,Z 389.258,A -85,B 0,C 180,E1 -29066.239,E2 -29066.239} C_VEL
LIN {X 0,Y 113.08,Z 389.241,A -85,B 0,C 180,E1 -29070,E2 -29070} C_VEL
LIN {X 0,Y 105.74,Z 389.153,A -85,B 0,C 180,E1 -29074.776,E2 -29074.776} C_VEL
LIN {X 0,Y 98.743,Z 388.233,A -85,B 0,C 180,E1 -29081.152,E2 -29081.152} C_VEL
LIN {X 0,Y 94.079,Z 386.721,A -85,B 0,C 180,E1 -29087.386,E2 -29087.386} C_VEL
LIN {X 0,Y 90.568,Z 384.012,A -85,B 0,C 180,E1 -29095.261,E2 -29095.261} C_VEL
LIN {X 0,Y 89.686,Z 382.503,A -85,B 0,C 180,E1 -29098.872,E2 -29098.872} C_VEL
LIN {X 0,Y 88.637,Z 381.024,A -85,B 0,C 180,E1 -29102.486,E2 -29102.486} C_VEL
LIN {X 0,Y 85.25,Z 377.491,A -85,B 0,C 180,E1 -29111.042,E2 -29111.042} C_VEL
LIN {X 0,Y 84.603,Z 374.976,A -85,B 0,C 180,E1 -29116.066,E2 -29116.066} C_VEL
LIN {X 0,Y 85.101,Z 373.481,A -85,B 0,C 180,E1 -29118.495,E2 -29118.495} C_VEL
LIN {X 0,Y 86.634,Z 369.428,A -85,B 0,C 180,E1 -29124.214,E2 -29124.214} C_VEL
LIN {X 0,Y 87.574,Z 366.428,A -85,B 0,C 180,E1 -29128.592,E2 -29128.592} C_VEL
LIN {X 0,Y 88.312,Z 363.234,A -85,B 0,C 180,E1 -29133.538,E2 -29133.538} C_VEL
LIN {X 0,Y 88.827,Z 360.097,A -85,B 0,C 180,E1 -29139.175,E2 -29139.175} C_VEL
LIN {X 0,Y 88.996,Z 358.874,A -85,B 0,C 180,E1 -29141.615,E2 -29141.615} C_VEL
LIN {X 0,Y 89.131,Z 357.076,A -85,B 0,C 180,E1 -29146.345,E2 -29146.345} C_VEL
LIN {X 0,Y 89.261,Z 355.846,A -85,B 0,C 180,E1 -29150.967,E2 -29150.967} C_VEL
LIN {X 0,Y 90.152,Z 354.173,A -85,B 0,C 180,E1 -29160.026,E2 -29160.026} C_VEL
LIN {X 0,Y 89.75,Z 355.106,A -85,B 0,C 180,E1 -29164.517,E2 -29164.517} C_VEL
LIN {X 0,Y 89.553,Z 356.35,A -85,B 0,C 180,E1 -29169.056,E2 -29169.056} C_VEL
LIN {X 0,Y 89.124,Z 358.257,A -85,B 0,C 180,E1 -29173.71,E2 -29173.71} C_VEL
LIN {X 0,Y 88.396,Z 361.025,A -85,B 0,C 180,E1 -29178.57,E2 -29178.57} C_VEL
LIN {X 0,Y 87.464,Z 363.844,A -85,B 0,C 180,E1 -29182.465,E2 -29182.465} C_VEL
LIN {X 0,Y 85.597,Z 366.688,A -85,B 0,C 180,E1 -29185.426,E2 -29185.426} C_VEL
LIN {X 0,Y 82.452,Z 370.767,A -85,B 0,C 180,E1 -29189.114,E2 -29189.114} C_VEL
LIN {X 0,Y 81.332,Z 371.939,A -85,B 0,C 180,E1 -29190.221,E2 -29190.221} C_VEL
LIN {X 0,Y 75.809,Z 376.441,A -85,B 0,C 180,E1 -29193.452,E2 -29193.452} C_VEL
LIN {X 0,Y 68.128,Z 381.937,A -85,B 0,C 180,E1 -29199.316,E2 -29199.316} C_VEL
LIN {X 0,Y 61.192,Z 386.265,A -85,B 0,C 180,E1 -29206.441,E2 -29206.441} C_VEL
LIN {X 0,Y 57.149,Z 388.634,A -85,B 0,C 180,E1 -29212.057,E2 -29212.057} C_VEL
LIN {X 0,Y 53.759,Z 390.438,A -85,B 0,C 180,E1 -29218.472,E2 -29218.472} C_VEL
LIN {X 0,Y 49.404,Z 392.905,A -85,B 0,C 180,E1 -29233.471,E2 -29233.471} C_VEL
LIN {X 0,Y 48.456,Z 393.504,A -85,B 0,C 180,E1 -29241.661,E2 -29241.661} C_VEL
LIN {X 0,Y 48.393,Z 393.668,A -85,B 0,C 180,E1 -29250,E2 -29250} C_VEL
LIN {X 0,Y 48.444,Z 393.503,A -85,B 0,C 180,E1 -29258.341,E2 -29258.341} C_VEL
LIN {X 0,Y 49.352,Z 392.903,A -85,B 0,C 180,E1 -29266.547,E2 -29266.547} C_VEL
LIN {X 0,Y 53.739,Z 390.438,A -85,B 0,C 180,E1 -29281.541,E2 -29281.541} C_VEL
LIN {X 0,Y 59.1,Z 387.482,A -85,B 0,C 180,E1 -29290.846,E2 -29290.846} C_VEL
LIN {X 0,Y 65.683,Z 383.49,A -85,B 0,C 180,E1 -29298.502,E2 -29298.502} C_VEL
LIN {X 0,Y 72.161,Z 379.109,A -85,B 0,C 180,E1 -29303.974,E2 -29303.974} C_VEL
LIN {X 0,Y 79.909,Z 373.094,A -85,B 0,C 180,E1 -29309.036,E2 -29309.036} C_VEL
LIN {X 0,Y 81.305,Z 371.938,A -85,B 0,C 180,E1 -29309.812,E2 -29309.812} C_VEL
LIN {X 0,Y 83.518,Z 369.492,A -85,B 0,C 180,E1 -29312.073,E2 -29312.073} C_VEL
LIN {X 0,Y 86.623,Z 365.201,A -85,B 0,C 180,E1 -29316.039,E2 -29316.039} C_VEL
LIN {X 0,Y 87.456,Z 363.85,A -85,B 0,C 180,E1 -29317.533,E2 -29317.533} C_VEL
LIN {X 0,Y 88.513,Z 360.491,A -85,B 0,C 180,E1 -29322.323,E2 -29322.323} C_VEL
LIN {X 0,Y 89.159,Z 358.223,A -85,B 0,C 180,E1 -29326.295,E2 -29326.295} C_VEL
LIN {X 0,Y 89.572,Z 356.332,A -85,B 0,C 180,E1 -29330.946,E2 -29330.946} C_VEL
LIN {X 0,Y 89.74,Z 355.118,A -85,B 0,C 180,E1 -29335.482,E2 -29335.482} C_VEL
LIN {X 0,Y 90.15,Z 354.175,A -85,B 0,C 180,E1 -29339.974,E2 -29339.974} C_VEL
LIN {X 0,Y 89.256,Z 355.85,A -85,B 0,C 180,E1 -29349.033,E2 -29349.033} C_VEL
LIN {X 0,Y 89.047,Z 357.155,A -85,B 0,C 180,E1 -29353.668,E2 -29353.668} C_VEL
LIN {X 0,Y 88.995,Z 358.975,A -85,B 0,C 180,E1 -29358.626,E2 -29358.626} C_VEL
LIN {X 0,Y 88.643,Z 361.483,A -85,B 0,C 180,E1 -29363.324,E2 -29363.324} C_VEL
LIN {X 0,Y 88.057,Z 364.524,A -85,B 0,C 180,E1 -29368.609,E2 -29368.609} C_VEL
LIN {X 0,Y 87,Z 368.483,A -85,B 0,C 180,E1 -29374.4,E2 -29374.4} C_VEL
LIN {X 0,Y 85.837,Z 371.639,A -85,B 0,C 180,E1 -29378.944,E2 -29378.944} C_VEL
LIN {X 0,Y 84.041,Z 375.579,A -85,B 0,C 180,E1 -29384.7,E2 -29384.7} C_VEL
LIN {X 0,Y 82.391,Z 380.485,A -85,B 0,C 180,E1 -29393.338,E2 -29393.338} C_VEL
LIN {X 0,Y 82.934,Z 384.245,A -85,B 0,C 180,E1 -29402.22,E2 -29402.22} C_VEL
LIN {X 0,Y 85.754,Z 386.961,A -85,B 0,C 180,E1 -29410.864,E2 -29410.864} C_VEL
LIN {X 0,Y 92.508,Z 389.04,A -85,B 0,C 180,E1 -29420.797,E2 -29420.797} C_VEL
LIN {X 0,Y 98.542,Z 389.56,A -85,B 0,C 180,E1 -29426.379,E2 -29426.379} C_VEL
LIN {X 0,Y 103.646,Z 389.5,A -85,B 0,C 180,E1 -29430,E2 -29430} C_VEL
LIN {X 0,Y 97.92,Z 389.512,A -85,B 0,C 180,E1 -29434.116,E2 -29434.116} C_VEL
LIN {X 0,Y 92.502,Z 389.043,A -85,B 0,C 180,E1 -29439.182,E2 -29439.182} C_VEL
LIN {X 0,Y 85.748,Z 386.961,A -85,B 0,C 180,E1 -29449.137,E2 -29449.137} C_VEL
LIN {X 0,Y 82.906,Z 384.246,A -85,B 0,C 180,E1 -29457.79,E2 -29457.79} C_VEL
LIN {X 0,Y 82.346,Z 380.487,A -85,B 0,C 180,E1 -29466.685,E2 -29466.685} C_VEL
LIN {X 0,Y 84.046,Z 375.579,A -85,B 0,C 180,E1 -29475.297,E2 -29475.297} C_VEL
LIN {X 0,Y 85.101,Z 373.481,A -85,B 0,C 180,E1 -29478.495,E2 -29478.495} C_VEL
LIN {X 0,Y 85.595,Z 371.998,A -85,B 0,C 180,E1 -29480.91,E2 -29480.91} C_VEL
LIN {X 0,Y 85.376,Z 370.126,A -85,B 0,C 180,E1 -29484.672,E2 -29484.672} C_VEL
LIN {X 0,Y 84.533,Z 368.581,A -85,B 0,C 180,E1 -29488.525,E2 -29488.525} C_VEL
LIN {X 0,Y 82.99,Z 365.65,A -85,B 0,C 180,E1 -29496.688,E2 -29496.688} C_VEL
LIN {X 0,Y 83.097,Z 364.501,A -85,B 0,C 180,E1 -29499.415,E2 -29499.415} C_VEL
LIN {X 0,Y 83.665,Z 362.227,A -85,B 0,C 180,E1 -29505.434,E2 -29505.434} C_VEL
LIN {X 0,Y 83.914,Z 360.845,A -85,B 0,C 180,E1 -29510.386,E2 -29510.386} C_VEL
LIN {X 0,Y 84.485,Z 359.616,A -85,B 0,C 180,E1 -29516.575,E2 -29516.575} C_VEL
LIN {X 0,Y 84.992,Z 359.148,A -85,B 0,C 180,E1 -29520.028,E2 -29520.028} C_VEL
LIN {X 0,Y 84.474,Z 360.092,A -85,B 0,C 180,E1 -29524.8,E2 -29524.8} C_VEL
LIN {X 0,Y 84.071,Z 361.481,A -85,B 0,C 180,E1 -29529.652,E2 -29529.652} C_VEL
LIN {X 0,Y 83.401,Z 363.624,A -85,B 0,C 180,E1 -29534.672,E2 -29534.672} C_VEL
LIN {X 0,Y 82.113,Z 366.439,A -85,B 0,C 180,E1 -29539.701,E2 -29539.701} C_VEL
LIN {X 0,Y 81.142,Z 367.887,A -85,B 0,C 180,E1 -29541.454,E2 -29541.454} C_VEL
LIN {X 0,Y 77.745,Z 371.728,A -85,B 0,C 180,E1 -29545.317,E2 -29545.317} C_VEL
LIN {X 0,Y 76.496,Z 372.899,A -85,B 0,C 180,E1 -29546.395,E2 -29546.395} C_VEL
LIN {X 0,Y 68.691,Z 378.563,A -85,B 0,C 180,E1 -29550.806,E2 -29550.806} C_VEL
LIN {X 0,Y 61.196,Z 383.295,A -85,B 0,C 180,E1 -29556.497,E2 -29556.497} C_VEL
LIN {X 0,Y 53.908,Z 387.287,A -85,B 0,C 180,E1 -29564.191,E2 -29564.191} C_VEL
LIN {X 0,Y 47.819,Z 390.243,A -85,B 0,C 180,E1 -29573.994,E2 -29573.994} C_VEL
LIN {X 0,Y 42.624,Z 392.709,A -85,B 0,C 180,E1 -29590.746,E2 -29590.746} C_VEL
LIN {X 0,Y 41.44,Z 393.309,A -85,B 0,C 180,E1 -29600.236,E2 -29600.236} C_VEL
LIN {X 0,Y 41.308,Z 393.474,A -85,B 0,C 180,E1 -29610,E2 -29610} C_VEL
LIN {X 0,Y 41.427,Z 393.308,A -85,B 0,C 180,E1 -29619.767,E2 -29619.767} C_VEL
LIN {X 0,Y 42.579,Z 392.708,A -85,B 0,C 180,E1 -29629.275,E2 -29629.275} C_VEL
LIN {X 0,Y 47.802,Z 390.242,A -85,B 0,C 180,E1 -29646.02,E2 -29646.02} C_VEL
LIN {X 0,Y 53.908,Z 387.287,A -85,B 0,C 180,E1 -29655.808,E2 -29655.808} C_VEL
LIN {X 0,Y 61.203,Z 383.295,A -85,B 0,C 180,E1 -29663.494,E2 -29663.494} C_VEL
LIN {X 0,Y 69.265,Z 378.202,A -85,B 0,C 180,E1 -29669.477,E2 -29669.477} C_VEL
LIN {X 0,Y 76.482,Z 372.898,A -85,B 0,C 180,E1 -29673.626,E2 -29673.626} C_VEL
LIN {X 0,Y 78.902,Z 370.55,A -85,B 0,C 180,E1 -29675.92,E2 -29675.92} C_VEL
LIN {X 0,Y 81.129,Z 367.893,A -85,B 0,C 180,E1 -29678.553,E2 -29678.553} C_VEL
LIN {X 0,Y 82.108,Z 366.439,A -85,B 0,C 180,E1 -29680.307,E2 -29680.307} C_VEL
LIN {X 0,Y 83.391,Z 363.632,A -85,B 0,C 180,E1 -29685.327,E2 -29685.327} C_VEL
LIN {X 0,Y 83.839,Z 362.419,A -85,B 0,C 180,E1 -29687.875,E2 -29687.875} C_VEL
LIN {X 0,Y 84.081,Z 361.472,A -85,B 0,C 180,E1 -29690.349,E2 -29690.349} C_VEL
LIN {X 0,Y 84.547,Z 359.919,A -85,B 0,C 180,E1 -29695.927,E2 -29695.927} C_VEL
LIN {X 0,Y 84.972,Z 359.167,A -85,B 0,C 180,E1 -29699.972,E2 -29699.972} C_VEL
LIN {X 0,Y 84.019,Z 360.376,A -85,B 0,C 180,E1 -29707.268,E2 -29707.268} C_VEL
LIN {X 0,Y 83.61,Z 362.275,A -85,B 0,C 180,E1 -29714.576,E2 -29714.576} C_VEL
LIN {X 0,Y 82.973,Z 364.854,A -85,B 0,C 180,E1 -29721.298,E2 -29721.298} C_VEL
LIN {X 0,Y 82.214,Z 367.773,A -85,B 0,C 180,E1 -29726.932,E2 -29726.932} C_VEL
LIN {X 0,Y 81.25,Z 370.186,A -85,B 0,C 180,E1 -29731.229,E2 -29731.229} C_VEL
LIN {X 0,Y 79.565,Z 373.972,A -85,B 0,C 180,E1 -29737.349,E2 -29737.349} C_VEL
LIN {X 0,Y 77.459,Z 377.643,A -85,B 0,C 180,E1 -29743.462,E2 -29743.462} C_VEL
LIN {X 0,Y 75.553,Z 382.168,A -85,B 0,C 180,E1 -29752.799,E2 -29752.799} C_VEL
LIN {X 0,Y 75.967,Z 385.552,A -85,B 0,C 180,E1 -29762.448,E2 -29762.448} C_VEL
LIN {X 0,Y 77.633,Z 387.198,A -85,B 0,C 180,E1 -29768.771,E2 -29768.771} C_VEL
LIN {X 0,Y 80.335,Z 388.432,A -85,B 0,C 180,E1 -29774.785,E2 -29774.785} C_VEL
LIN {X 0,Y 85.182,Z 389.441,A -85,B 0,C 180,E1 -29781.701,E2 -29781.701} C_VEL
LIN {X 0,Y 94.339,Z 389.755,A -85,B 0,C 180,E1 -29790,E2 -29790} C_VEL
LIN {X 0,Y 85.178,Z 389.444,A -85,B 0,C 180,E1 -29798.281,E2 -29798.281} C_VEL
LIN {X 0,Y 80.168,Z 388.388,A -85,B 0,C 180,E1 -29805.474,E2 -29805.474} C_VEL
LIN {X 0,Y 76.764,Z 386.529,A -85,B 0,C 180,E1 -29813.803,E2 -29813.803} C_VEL
LIN {X 0,Y 75.379,Z 383.692,A -85,B 0,C 180,E1 -29823.016,E2 -29823.016} C_VEL
LIN {X 0,Y 75.923,Z 380.712,A -85,B 0,C 180,E1 -29830.387,E2 -29830.387} C_VEL
LIN {X 0,Y 78.303,Z 376.108,A -85,B 0,C 180,E1 -29839.067,E2 -29839.067} C_VEL
LIN {X 0,Y 80.048,Z 372.984,A -85,B 0,C 180,E1 -29844.302,E2 -29844.302} C_VEL
LIN {X 0,Y 81.438,Z 369.689,A -85,B 0,C 180,E1 -29849.652,E2 -29849.652} C_VEL
LIN {X 0,Y 82.48,Z 366.797,A -85,B 0,C 180,E1 -29854.816,E2 -29854.816} C_VEL
LIN {X 0,Y 83.097,Z 364.501,A -85,B 0,C 180,E1 -29859.415,E2 -29859.415} C_VEL
LIN {X 0,Y 82.817,Z 363.825,A -85,B 0,C 180,E1 -29862.054,E2 -29862.054} C_VEL
LIN {X 0,Y 81.747,Z 363.878,A -85,B 0,C 180,E1 -29864.725,E2 -29864.725} C_VEL
LIN {X 0,Y 78.891,Z 364.833,A -85,B 0,C 180,E1 -29871.241,E2 -29871.241} C_VEL
LIN {X 0,Y 78.687,Z 364.699,A -85,B 0,C 180,E1 -29874.216,E2 -29874.216} C_VEL
LIN {X 0,Y 79.587,Z 363.903,A -85,B 0,C 180,E1 -29880.03,E2 -29880.03} C_VEL
LIN {X 0,Y 78.92,Z 364.863,A -85,B 0,C 180,E1 -29885.139,E2 -29885.139} C_VEL
LIN {X 0,Y 78.31,Z 366.281,A -85,B 0,C 180,E1 -29890.37,E2 -29890.37} C_VEL
LIN {X 0,Y 77.799,Z 367.353,A -85,B 0,C 180,E1 -29893.082,E2 -29893.082} C_VEL
LIN {X 0,Y 76.455,Z 369.748,A -85,B 0,C 180,E1 -29897.65,E2 -29897.65} C_VEL
LIN {X 0,Y 73.411,Z 372.689,A -85,B 0,C 180,E1 -29901.031,E2 -29901.031} C_VEL
LIN {X 0,Y 72.049,Z 373.859,A -85,B 0,C 180,E1 -29902.082,E2 -29902.082} C_VEL
LIN {X 0,Y 62.983,Z 379.882,A -85,B 0,C 180,E1 -29906.79,E2 -29906.79} C_VEL
LIN {X 0,Y 54.452,Z 384.63,A -85,B 0,C 180,E1 -29912.973,E2 -29912.973} C_VEL
LIN {X 0,Y 46.739,Z 388.243,A -85,B 0,C 180,E1 -29921.252,E2 -29921.252} C_VEL
LIN {X 0,Y 42.255,Z 390.047,A -85,B 0,C 180,E1 -29928.296,E2 -29928.296} C_VEL
LIN {X 0,Y 35.984,Z 392.514,A -85,B 0,C 180,E1 -29947.008,E2 -29947.008} C_VEL
LIN {X 0,Y 34.445,Z 393.114,A -85,B 0,C 180,E1 -29958.227,E2 -29958.227} C_VEL
LIN {X 0,Y 34.194,Z 393.279,A -85,B 0,C 180,E1 -29970,E2 -29970} C_VEL
LIN {X 0,Y 34.431,Z 393.113,A -85,B 0,C 180,E1 -29981.777,E2 -29981.777} C_VEL
LIN {X 0,Y 35.919,Z 392.512,A -85,B 0,C 180,E1 -29993.036,E2 -29993.036} C_VEL
LIN {X 0,Y 42.241,Z 390.046,A -85,B 0,C 180,E1 -30011.721,E2 -30011.721} C_VEL
LIN {X 0,Y 49.205,Z 387.092,A -85,B 0,C 180,E1 -30021.771,E2 -30021.771} C_VEL
LIN {X 0,Y 57.257,Z 383.1,A -85,B 0,C 180,E1 -30029.225,E2 -30029.225} C_VEL
LIN {X 0,Y 66.235,Z 377.801,A -85,B 0,C 180,E1 -30035.026,E2 -30035.026} C_VEL
LIN {X 0,Y 72.044,Z 373.858,A -85,B 0,C 180,E1 -30037.929,E2 -30037.929} C_VEL
LIN {X 0,Y 74.668,Z 371.508,A -85,B 0,C 180,E1 -30040.256,E2 -30040.256} C_VEL
LIN {X 0,Y 76.446,Z 369.753,A -85,B 0,C 180,E1 -30042.354,E2 -30042.354} C_VEL
LIN {X 0,Y 77.774,Z 367.373,A -85,B 0,C 180,E1 -30046.913,E2 -30046.913} C_VEL
LIN {X 0,Y 78.413,Z 366.04,A -85,B 0,C 180,E1 -30050.362,E2 -30050.362} C_VEL
LIN {X 0,Y 78.932,Z 364.853,A -85,B 0,C 180,E1 -30054.862,E2 -30054.862} C_VEL
LIN {X 0,Y 79.569,Z 363.917,A -85,B 0,C 180,E1 -30059.97,E2 -30059.97} C_VEL
LIN {X 0,Y 78.529,Z 364.916,A -85,B 0,C 180,E1 -30066.954,E2 -30066.954} C_VEL
LIN {X 0,Y 78.209,Z 365.579,A -85,B 0,C 180,E1 -30070.322,E2 -30070.322} C_VEL
LIN {X 0,Y 77.458,Z 367.998,A -85,B 0,C 180,E1 -30078.483,E2 -30078.483} C_VEL
LIN {X 0,Y 76.391,Z 370.422,A -85,B 0,C 180,E1 -30084.418,E2 -30084.418} C_VEL
LIN {X 0,Y 74.866,Z 373.559,A -85,B 0,C 180,E1 -30090.56,E2 -30090.56} C_VEL
LIN {X 0,Y 72.719,Z 376.849,A -85,B 0,C 180,E1 -30096.867,E2 -30096.867} C_VEL
LIN {X 0,Y 69.152,Z 382.394,A -85,B 0,C 180,E1 -30108.656,E2 -30108.656} C_VEL
LIN {X 0,Y 68.578,Z 385.784,A -85,B 0,C 180,E1 -30119.176,E2 -30119.176} C_VEL
LIN {X 0,Y 69.632,Z 387.435,A -85,B 0,C 180,E1 -30126.189,E2 -30126.189} C_VEL
LIN {X 0,Y 75.357,Z 389.576,A -85,B 0,C 180,E1 -30139.25,E2 -30139.25} C_VEL
LIN {X 0,Y 79.754,Z 390.011,A -85,B 0,C 180,E1 -30144.945,E2 -30144.945} C_VEL
LIN {X 0,Y 85.127,Z 390.008,A -85,B 0,C 180,E1 -30150,E2 -30150} C_VEL
LIN {X 0,Y 77.877,Z 389.843,A -85,B 0,C 180,E1 -30157.207,E2 -30157.207} C_VEL
LIN {X 0,Y 71.953,Z 388.671,A -85,B 0,C 180,E1 -30167.039,E2 -30167.039} C_VEL
LIN {X 0,Y 69.462,Z 387.273,A -85,B 0,C 180,E1 -30174.502,E2 -30174.502} C_VEL
LIN {X 0,Y 68.425,Z 384.576,A -85,B 0,C 180,E1 -30184.812,E2 -30184.812} C_VEL
LIN {X 0,Y 69.884,Z 380.936,A -85,B 0,C 180,E1 -30194.745,E2 -30194.745} C_VEL
